LIN {X 0,Y 587.697,Z 859.31,A -85,B 0,C 180,E1 8837.447,E2 8837.447} C_VEL
LIN {X 0,Y 587.589,Z 859.31,A -85,B 0,C 180,E1 8842.753,E2 8842.753} C_VEL
LIN {X 0,Y 587.459,Z 859.31,A -85,B 0,C 180,E1 8847.659,E2 8847.659} C_VEL
LIN {X 0,Y 587.346,Z 859.31,A -85,B 0,C 180,E1 8852.797,E2 8852.797} C_VEL
LIN {X 0,Y 587.19,Z 859.31,A -85,B 0,C 180,E1 8858.258,E2 8858.258} C_VEL
LIN {X 0,Y 587.185,Z 859.31,A -85,B 0,C 180,E1 8864.156,E2 8864.156} C_VEL
LIN {X 0,Y 587.224,Z 859.31,A -85,B 0,C 180,E1 8869.826,E2 8869.826} C_VEL
LIN {X 0,Y 587.363,Z 859.919,A -85,B 0,C 180,E1 8871.339,E2 8871.339} C_VEL
LIN {X 0,Y 612.284,Z 916.303,A -85,B 0,C 180,E1 8873.785,E2 8873.785} C_VEL
LIN {X 0,Y 612.06,Z 926.776,A -85,B 0,C 180,E1 8873.959,E2 8873.959} C_VEL
LIN {X 0,Y 608.088,Z 943.76,A -85,B 0,C 180,E1 8874.115,E2 8874.115} C_VEL
LIN {X 0,Y 603.502,Z 960.575,A -85,B 0,C 180,E1 8874.323,E2 8874.323} C_VEL
LIN {X 0,Y 600.339,Z 1006.753,A -85,B 0,C 180,E1 8875.92,E2 8875.92} C_VEL
LIN {X 0,Y 596.482,Z 1051.642,A -85,B 0,C 180,E1 8878.158,E2 8878.158} C_VEL
LIN {X 0,Y 592.489,Z 1093.023,A -85,B 0,C 180,E1 8880.927,E2 8880.927} C_VEL
LIN {X 0,Y 588.871,Z 1128.661,A -85,B 0,C 180,E1 8884.059,E2 8884.059} C_VEL
LIN {X 0,Y 585.696,Z 1159.357,A -85,B 0,C 180,E1 8887.567,E2 8887.567} C_VEL
LIN {X 0,Y 583.284,Z 1184.333,A -85,B 0,C 180,E1 8891.257,E2 8891.257} C_VEL
LIN {X 0,Y 581.725,Z 1204.991,A -85,B 0,C 180,E1 8895.287,E2 8895.287} C_VEL
LIN {X 0,Y 580.827,Z 1221.162,A -85,B 0,C 180,E1 8899.857,E2 8899.857} C_VEL
LIN {X 0,Y 580.497,Z 1230.457,A -85,B 0,C 180,E1 8904.006,E2 8904.006} C_VEL
LIN {X 0,Y 580.504,Z 1235.164,A -85,B 0,C 180,E1 8908.504,E2 8908.504} C_VEL
LIN {X 0,Y 580.466,Z 1234.213,A -85,B 0,C 180,E1 8912.993,E2 8912.993} C_VEL
LIN {X 0,Y 580.544,Z 1229.327,A -85,B 0,C 180,E1 8916.683,E2 8916.683} C_VEL
LIN {X 0,Y 580.955,Z 1217.72,A -85,B 0,C 180,E1 8921.281,E2 8921.281} C_VEL
LIN {X 0,Y 582.016,Z 1201.38,A -85,B 0,C 180,E1 8925.504,E2 8925.504} C_VEL
LIN {X 0,Y 583.753,Z 1179.913,A -85,B 0,C 180,E1 8929.471,E2 8929.471} C_VEL
LIN {X 0,Y 586.43,Z 1151.644,A -85,B 0,C 180,E1 8933.414,E2 8933.414} C_VEL
LIN {X 0,Y 590.023,Z 1117.476,A -85,B 0,C 180,E1 8937.016,E2 8937.016} C_VEL
LIN {X 0,Y 594.013,Z 1078.354,A -85,B 0,C 180,E1 8940.148,E2 8940.148} C_VEL
LIN {X 0,Y 598.073,Z 1034.825,A -85,B 0,C 180,E1 8942.765,E2 8942.765} C_VEL
LIN {X 0,Y 601.694,Z 989.173,A -85,B 0,C 180,E1 8944.77,E2 8944.77} C_VEL
LIN {X 0,Y 604.598,Z 941.328,A -85,B 0,C 180,E1 8946.155,E2 8946.155} C_VEL
LIN {X 0,Y 605.195,Z 918.263,A -85,B 0,C 180,E1 8946.6,E2 8946.6} C_VEL
LIN {X 0,Y 583.541,Z 869.006,A -85,B 0,C 180,E1 8948.782,E2 8948.782} C_VEL
LIN {X 0,Y 579.403,Z 859.31,A -85,B 0,C 180,E1 8949.238,E2 8949.238} C_VEL
LIN {X 0,Y 579.376,Z 859.31,A -85,B 0,C 180,E1 8955.089,E2 8955.089} C_VEL
LIN {X 0,Y 579.271,Z 859.31,A -85,B 0,C 180,E1 8961.121,E2 8961.121} C_VEL
LIN {X 0,Y 579.379,Z 859.31,A -85,B 0,C 180,E1 8966.816,E2 8966.816} C_VEL
LIN {X 0,Y 579.578,Z 859.31,A -85,B 0,C 180,E1 8972.738,E2 8972.738} C_VEL
LIN {X 0,Y 579.689,Z 859.31,A -85,B 0,C 180,E1 8978.537,E2 8978.537} C_VEL
LIN {X 0,Y 579.76,Z 859.31,A -85,B 0,C 180,E1 8983.294,E2 8983.294} C_VEL
LIN {X 0,Y 579.901,Z 859.31,A -85,B 0,C 180,E1 8989.461,E2 8989.461} C_VEL
LIN {X 0,Y 580.104,Z 859.31,A -85,B 0,C 180,E1 8994.002,E2 8994.002} C_VEL
LIN {X 0,Y 580.244,Z 859.31,A -85,B 0,C 180,E1 8998.502,E2 8998.502} C_VEL
LIN {X 0,Y 580.215,Z 859.31,A -85,B 0,C 180,E1 9002.991,E2 9002.991} C_VEL
LIN {X 0,Y 580.045,Z 859.31,A -85,B 0,C 180,E1 9007.501,E2 9007.501} C_VEL
LIN {X 0,Y 579.905,Z 859.31,A -85,B 0,C 180,E1 9012.061,E2 9012.061} C_VEL
LIN {X 0,Y 579.803,Z 859.31,A -85,B 0,C 180,E1 9016.7,E2 9016.7} C_VEL
LIN {X 0,Y 579.663,Z 859.31,A -85,B 0,C 180,E1 9021.459,E2 9021.459} C_VEL
LIN {X 0,Y 579.514,Z 859.31,A -85,B 0,C 180,E1 9027.25,E2 9027.25} C_VEL
LIN {X 0,Y 579.386,Z 859.31,A -85,B 0,C 180,E1 9033.301,E2 9033.301} C_VEL
LIN {X 0,Y 579.282,Z 859.31,A -85,B 0,C 180,E1 9038.873,E2 9038.873} C_VEL
LIN {X 0,Y 579.235,Z 859.31,A -85,B 0,C 180,E1 9045.063,E2 9045.063} C_VEL
LIN {X 0,Y 579.333,Z 859.31,A -85,B 0,C 180,E1 9051.117,E2 9051.117} C_VEL
LIN {X 0,Y 579.475,Z 859.947,A -85,B 0,C 180,E1 9057.039,E2 9057.039} C_VEL
LIN {X 0,Y 604.152,Z 909.899,A -85,B 0,C 180,E1 9059.386,E2 9059.386} C_VEL
LIN {X 0,Y 603.053,Z 971.893,A -85,B 0,C 180,E1 9060.257,E2 9060.257} C_VEL
LIN {X 0,Y 600.509,Z 1012.044,A -85,B 0,C 180,E1 9061.399,E2 9061.399} C_VEL
LIN {X 0,Y 596.94,Z 1050.359,A -85,B 0,C 180,E1 9063.118,E2 9063.118} C_VEL
LIN {X 0,Y 592.943,Z 1085.359,A -85,B 0,C 180,E1 9065.354,E2 9065.354} C_VEL
LIN {X 0,Y 588.966,Z 1116.703,A -85,B 0,C 180,E1 9068.072,E2 9068.072} C_VEL
LIN {X 0,Y 585.696,Z 1143.269,A -85,B 0,C 180,E1 9071.138,E2 9071.138} C_VEL
LIN {X 0,Y 583.07,Z 1166.127,A -85,B 0,C 180,E1 9074.658,E2 9074.658} C_VEL
LIN {X 0,Y 581.532,Z 1183.649,A -85,B 0,C 180,E1 9078.35,E2 9078.35} C_VEL
LIN {X 0,Y 580.757,Z 1196.752,A -85,B 0,C 180,E1 9082.386,E2 9082.386} C_VEL
LIN {X 0,Y 580.526,Z 1203,A -85,B 0,C 180,E1 9085.509,E2 9085.509} C_VEL
LIN {X 0,Y 580.388,Z 1205.958,A -85,B 0,C 180,E1 9088.504,E2 9088.504} C_VEL
LIN {X 0,Y 580.489,Z 1205.894,A -85,B 0,C 180,E1 9091.496,E2 9091.496} C_VEL
LIN {X 0,Y 580.614,Z 1201.69,A -85,B 0,C 180,E1 9095.241,E2 9095.241} C_VEL
LIN {X 0,Y 580.972,Z 1191.508,A -85,B 0,C 180,E1 9099.382,E2 9099.382} C_VEL
LIN {X 0,Y 582.164,Z 1175.966,A -85,B 0,C 180,E1 9103.334,E2 9103.334} C_VEL
LIN {X 0,Y 584.19,Z 1155.887,A -85,B 0,C 180,E1 9106.966,E2 9106.966} C_VEL
LIN {X 0,Y 587.292,Z 1130.212,A -85,B 0,C 180,E1 9110.385,E2 9110.385} C_VEL
LIN {X 0,Y 591.008,Z 1100.781,A -85,B 0,C 180,E1 9113.316,E2 9113.316} C_VEL
LIN {X 0,Y 595.002,Z 1067.95,A -85,B 0,C 180,E1 9115.756,E2 9115.756} C_VEL
LIN {X 0,Y 598.679,Z 1033,A -85,B 0,C 180,E1 9117.652,E2 9117.652} C_VEL
LIN {X 0,Y 601.636,Z 995.563,A -85,B 0,C 180,E1 9119.055,E2 9119.055} C_VEL
LIN {X 0,Y 603.581,Z 956.066,A -85,B 0,C 180,E1 9119.942,E2 9119.942} C_VEL
LIN {X 0,Y 603.684,Z 908.974,A -85,B 0,C 180,E1 9120.562,E2 9120.562} C_VEL
LIN {X 0,Y 579.497,Z 860.059,A -85,B 0,C 180,E1 9122.861,E2 9122.861} C_VEL
LIN {X 0,Y 579.373,Z 859.31,A -85,B 0,C 180,E1 9128.337,E2 9128.337} C_VEL
LIN {X 0,Y 579.233,Z 859.31,A -85,B 0,C 180,E1 9132.924,E2 9132.924} C_VEL
LIN {X 0,Y 579.287,Z 859.31,A -85,B 0,C 180,E1 9139.176,E2 9139.176} C_VEL
LIN {X 0,Y 579.351,Z 859.31,A -85,B 0,C 180,E1 9144.885,E2 9144.885} C_VEL
LIN {X 0,Y 579.416,Z 859.31,A -85,B 0,C 180,E1 9150.217,E2 9150.217} C_VEL
LIN {X 0,Y 579.59,Z 859.31,A -85,B 0,C 180,E1 9155.282,E2 9155.282} C_VEL
LIN {X 0,Y 579.568,Z 859.31,A -85,B 0,C 180,E1 9160.259,E2 9160.259} C_VEL
LIN {X 0,Y 579.713,Z 859.31,A -85,B 0,C 180,E1 9166.4,E2 9166.4} C_VEL
LIN {X 0,Y 580.093,Z 859.31,A -85,B 0,C 180,E1 9172.169,E2 9172.169} C_VEL
LIN {X 0,Y 580.271,Z 859.31,A -85,B 0,C 180,E1 9177.009,E2 9177.009} C_VEL
LIN {X 0,Y 580.392,Z 859.31,A -85,B 0,C 180,E1 9181.498,E2 9181.498} C_VEL
LIN {X 0,Y 580.005,Z 859.31,A -85,B 0,C 180,E1 9186.893,E2 9186.893} C_VEL
LIN {X 0,Y 579.884,Z 859.31,A -85,B 0,C 180,E1 9192.065,E2 9192.065} C_VEL
LIN {X 0,Y 579.807,Z 859.31,A -85,B 0,C 180,E1 9196.705,E2 9196.705} C_VEL
LIN {X 0,Y 579.692,Z 859.31,A -85,B 0,C 180,E1 9201.463,E2 9201.463} C_VEL
LIN {X 0,Y 579.545,Z 859.31,A -85,B 0,C 180,E1 9207.255,E2 9207.255} C_VEL
LIN {X 0,Y 579.385,Z 859.31,A -85,B 0,C 180,E1 9213.306,E2 9213.306} C_VEL
LIN {X 0,Y 579.262,Z 859.31,A -85,B 0,C 180,E1 9218.88,E2 9218.88} C_VEL
LIN {X 0,Y 579.222,Z 859.31,A -85,B 0,C 180,E1 9225.062,E2 9225.062} C_VEL
LIN {X 0,Y 579.378,Z 859.31,A -85,B 0,C 180,E1 9230.754,E2 9230.754} C_VEL
LIN {X 0,Y 599.876,Z 906.09,A -85,B 0,C 180,E1 9232.87,E2 9232.87} C_VEL
LIN {X 0,Y 605.474,Z 920.812,A -85,B 0,C 180,E1 9233.461,E2 9233.461} C_VEL
LIN {X 0,Y 603.502,Z 960.575,A -85,B 0,C 180,E1 9234.323,E2 9234.323} C_VEL
LIN {X 0,Y 594.723,Z 991.691,A -85,B 0,C 180,E1 9234.944,E2 9234.944} C_VEL
LIN {X 0,Y 594.491,Z 993.669,A -85,B 0,C 180,E1 9235.019,E2 9235.019} C_VEL
LIN {X 0,Y 590.821,Z 1037.331,A -85,B 0,C 180,E1 9237.016,E2 9237.016} C_VEL
LIN {X 0,Y 586.644,Z 1078.873,A -85,B 0,C 180,E1 9239.595,E2 9239.595} C_VEL
LIN {X 0,Y 582.519,Z 1117.313,A -85,B 0,C 180,E1 9242.711,E2 9242.711} C_VEL
LIN {X 0,Y 578.817,Z 1151.567,A -85,B 0,C 180,E1 9246.357,E2 9246.357} C_VEL
LIN {X 0,Y 576.12,Z 1178.982,A -85,B 0,C 180,E1 9250.202,E2 9250.202} C_VEL
LIN {X 0,Y 574.243,Z 1200.385,A -85,B 0,C 180,E1 9254.154,E2 9254.154} C_VEL
LIN {X 0,Y 573.197,Z 1216.803,A -85,B 0,C 180,E1 9258.266,E2 9258.266} C_VEL
LIN {X 0,Y 572.66,Z 1227.634,A -85,B 0,C 180,E1 9262.397,E2 9262.397} C_VEL
LIN {X 0,Y 572.539,Z 1232.645,A -85,B 0,C 180,E1 9265.446,E2 9265.446} C_VEL
LIN {X 0,Y 572.567,Z 1235.5,A -85,B 0,C 180,E1 9270,E2 9270} C_VEL
LIN {X 0,Y 572.544,Z 1232.646,A -85,B 0,C 180,E1 9274.554,E2 9274.554} C_VEL
LIN {X 0,Y 572.685,Z 1226.068,A -85,B 0,C 180,E1 9278.368,E2 9278.368} C_VEL
LIN {X 0,Y 573.34,Z 1213.755,A -85,B 0,C 180,E1 9282.594,E2 9282.594} C_VEL
LIN {X 0,Y 574.504,Z 1196.74,A -85,B 0,C 180,E1 9286.612,E2 9286.612} C_VEL
LIN {X 0,Y 576.593,Z 1172.554,A -85,B 0,C 180,E1 9290.809,E2 9290.809} C_VEL
LIN {X 0,Y 579.67,Z 1143.649,A -85,B 0,C 180,E1 9294.568,E2 9294.568} C_VEL
LIN {X 0,Y 583.082,Z 1111.739,A -85,B 0,C 180,E1 9297.785,E2 9297.785} C_VEL
LIN {X 0,Y 587.072,Z 1074.285,A -85,B 0,C 180,E1 9300.722,E2 9300.722} C_VEL
LIN {X 0,Y 591.139,Z 1033.204,A -85,B 0,C 180,E1 9303.206,E2 9303.206} C_VEL
LIN {X 0,Y 594.921,Z 988.204,A -85,B 0,C 180,E1 9305.191,E2 9305.191} C_VEL
LIN {X 0,Y 597.93,Z 940.993,A -85,B 0,C 180,E1 9306.564,E2 9306.564} C_VEL
LIN {X 0,Y 598.169,Z 920.224,A -85,B 0,C 180,E1 9306.997,E2 9306.997} C_VEL
LIN {X 0,Y 577.934,Z 873.583,A -85,B 0,C 180,E1 9309.102,E2 9309.102} C_VEL
LIN {X 0,Y 571.434,Z 859.31,A -85,B 0,C 180,E1 9309.855,E2 9309.855} C_VEL
LIN {X 0,Y 571.382,Z 859.31,A -85,B 0,C 180,E1 9315.728,E2 9315.728} C_VEL
LIN {X 0,Y 571.327,Z 859.31,A -85,B 0,C 180,E1 9320.476,E2 9320.476} C_VEL
LIN {X 0,Y 571.383,Z 859.31,A -85,B 0,C 180,E1 9326.165,E2 9326.165} C_VEL
LIN {X 0,Y 571.588,Z 859.31,A -85,B 0,C 180,E1 9331.504,E2 9331.504} C_VEL
LIN {X 0,Y 571.752,Z 859.31,A -85,B 0,C 180,E1 9336.58,E2 9336.58} C_VEL
LIN {X 0,Y 571.821,Z 859.31,A -85,B 0,C 180,E1 9342.549,E2 9342.549} C_VEL
LIN {X 0,Y 571.928,Z 859.31,A -85,B 0,C 180,E1 9348.606,E2 9348.606} C_VEL
LIN {X 0,Y 572.205,Z 859.31,A -85,B 0,C 180,E1 9353.919,E2 9353.919} C_VEL
LIN {X 0,Y 572.342,Z 859.31,A -85,B 0,C 180,E1 9358.481,E2 9358.481} C_VEL
LIN {X 0,Y 572.314,Z 859.31,A -85,B 0,C 180,E1 9363.033,E2 9363.033} C_VEL
LIN {X 0,Y 572.127,Z 859.31,A -85,B 0,C 180,E1 9367.606,E2 9367.606} C_VEL
LIN {X 0,Y 571.984,Z 859.31,A -85,B 0,C 180,E1 9372.23,E2 9372.23} C_VEL
LIN {X 0,Y 571.829,Z 859.31,A -85,B 0,C 180,E1 9377.453,E2 9377.453} C_VEL
LIN {X 0,Y 571.699,Z 859.31,A -85,B 0,C 180,E1 9383.418,E2 9383.418} C_VEL
LIN {X 0,Y 571.54,Z 859.31,A -85,B 0,C 180,E1 9388.966,E2 9388.966} C_VEL
LIN {X 0,Y 571.392,Z 859.31,A -85,B 0,C 180,E1 9394.705,E2 9394.705} C_VEL
LIN {X 0,Y 571.309,Z 859.31,A -85,B 0,C 180,E1 9399.721,E2 9399.721} C_VEL
LIN {X 0,Y 571.258,Z 859.31,A -85,B 0,C 180,E1 9405.722,E2 9405.722} C_VEL
LIN {X 0,Y 571.349,Z 859.31,A -85,B 0,C 180,E1 9410.468,E2 9410.468} C_VEL
LIN {X 0,Y 571.475,Z 859.31,A -85,B 0,C 180,E1 9416.435,E2 9416.435} C_VEL
LIN {X 0,Y 578.232,Z 873.768,A -85,B 0,C 180,E1 9417.136,E2 9417.136} C_VEL
LIN {X 0,Y 597.673,Z 913.926,A -85,B 0,C 180,E1 9419.013,E2 9419.013} C_VEL
LIN {X 0,Y 596.487,Z 971.573,A -85,B 0,C 180,E1 9419.832,E2 9419.832} C_VEL
LIN {X 0,Y 593.767,Z 1012.202,A -85,B 0,C 180,E1 9420.996,E2 9420.996} C_VEL
LIN {X 0,Y 590.145,Z 1049.593,A -85,B 0,C 180,E1 9422.68,E2 9422.68} C_VEL
LIN {X 0,Y 585.912,Z 1084.949,A -85,B 0,C 180,E1 9424.945,E2 9424.945} C_VEL
LIN {X 0,Y 581.693,Z 1116.6,A -85,B 0,C 180,E1 9427.708,E2 9427.708} C_VEL
LIN {X 0,Y 578.142,Z 1143.832,A -85,B 0,C 180,E1 9430.887,E2 9430.887} C_VEL
LIN {X 0,Y 575.352,Z 1166.873,A -85,B 0,C 180,E1 9434.493,E2 9434.493} C_VEL
LIN {X 0,Y 573.743,Z 1184.091,A -85,B 0,C 180,E1 9438.189,E2 9438.189} C_VEL
LIN {X 0,Y 573.01,Z 1195.446,A -85,B 0,C 180,E1 9441.637,E2 9441.637} C_VEL
LIN {X 0,Y 572.663,Z 1203.237,A -85,B 0,C 180,E1 9445.447,E2 9445.447} C_VEL
LIN {X 0,Y 572.506,Z 1206.164,A -85,B 0,C 180,E1 9448.484,E2 9448.484} C_VEL
LIN {X 0,Y 572.62,Z 1206.103,A -85,B 0,C 180,E1 9451.517,E2 9451.517} C_VEL
LIN {X 0,Y 572.731,Z 1201.943,A -85,B 0,C 180,E1 9455.313,E2 9455.313} C_VEL
LIN {X 0,Y 573.136,Z 1191.887,A -85,B 0,C 180,E1 9459.511,E2 9459.511} C_VEL
LIN {X 0,Y 574.369,Z 1177.169,A -85,B 0,C 180,E1 9463.371,E2 9463.371} C_VEL
LIN {X 0,Y 576.586,Z 1156.417,A -85,B 0,C 180,E1 9467.197,E2 9467.197} C_VEL
LIN {X 0,Y 579.852,Z 1130.793,A -85,B 0,C 180,E1 9470.658,E2 9470.658} C_VEL
LIN {X 0,Y 583.768,Z 1101.465,A -85,B 0,C 180,E1 9473.623,E2 9473.623} C_VEL
LIN {X 0,Y 587.928,Z 1068.798,A -85,B 0,C 180,E1 9476.089,E2 9476.089} C_VEL
LIN {X 0,Y 591.882,Z 1033.144,A -85,B 0,C 180,E1 9478.046,E2 9478.046} C_VEL
LIN {X 0,Y 594.997,Z 995.399,A -85,B 0,C 180,E1 9479.473,E2 9479.473} C_VEL
LIN {X 0,Y 597.042,Z 954.642,A -85,B 0,C 180,E1 9480.384,E2 9480.384} C_VEL
LIN {X 0,Y 597.195,Z 911.71,A -85,B 0,C 180,E1 9480.953,E2 9480.953} C_VEL
LIN {X 0,Y 571.691,Z 860.878,A -85,B 0,C 180,E1 9483.428,E2 9483.428} C_VEL
LIN {X 0,Y 571.494,Z 859.31,A -85,B 0,C 180,E1 9483.51,E2 9483.51} C_VEL
LIN {X 0,Y 571.468,Z 859.31,A -85,B 0,C 180,E1 9487.58,E2 9487.58} C_VEL
LIN {X 0,Y 571.272,Z 859.31,A -85,B 0,C 180,E1 9493.602,E2 9493.602} C_VEL
LIN {X 0,Y 571.286,Z 859.31,A -85,B 0,C 180,E1 9498.479,E2 9498.479} C_VEL
LIN {X 0,Y 571.455,Z 859.31,A -85,B 0,C 180,E1 9504.326,E2 9504.326} C_VEL
LIN {X 0,Y 571.52,Z 859.31,A -85,B 0,C 180,E1 9509.763,E2 9509.763} C_VEL
LIN {X 0,Y 571.638,Z 859.31,A -85,B 0,C 180,E1 9514.914,E2 9514.914} C_VEL
LIN {X 0,Y 571.662,Z 859.31,A -85,B 0,C 180,E1 9519.851,E2 9519.851} C_VEL
LIN {X 0,Y 571.812,Z 859.31,A -85,B 0,C 180,E1 9526.208,E2 9526.208} C_VEL
LIN {X 0,Y 572.191,Z 859.31,A -85,B 0,C 180,E1 9532.184,E2 9532.184} C_VEL
LIN {X 0,Y 572.364,Z 859.31,A -85,B 0,C 180,E1 9536.968,E2 9536.968} C_VEL
LIN {X 0,Y 572.486,Z 859.31,A -85,B 0,C 180,E1 9541.518,E2 9541.518} C_VEL
LIN {X 0,Y 572.229,Z 859.31,A -85,B 0,C 180,E1 9546.081,E2 9546.081} C_VEL
LIN {X 0,Y 571.968,Z 859.31,A -85,B 0,C 180,E1 9552.235,E2 9552.235} C_VEL
LIN {X 0,Y 571.863,Z 859.31,A -85,B 0,C 180,E1 9557.463,E2 9557.463} C_VEL
LIN {X 0,Y 571.725,Z 859.31,A -85,B 0,C 180,E1 9563.421,E2 9563.421} C_VEL
LIN {X 0,Y 571.568,Z 859.31,A -85,B 0,C 180,E1 9568.97,E2 9568.97} C_VEL
LIN {X 0,Y 571.396,Z 859.31,A -85,B 0,C 180,E1 9574.705,E2 9574.705} C_VEL
LIN {X 0,Y 571.306,Z 859.31,A -85,B 0,C 180,E1 9579.72,E2 9579.72} C_VEL
LIN {X 0,Y 571.249,Z 859.31,A -85,B 0,C 180,E1 9585.729,E2 9585.729} C_VEL
LIN {X 0,Y 571.412,Z 859.519,A -85,B 0,C 180,E1 9590.2,E2 9590.2} C_VEL
LIN {X 0,Y 591.691,Z 904.574,A -85,B 0,C 180,E1 9592.325,E2 9592.325} C_VEL
LIN {X 0,Y 598.794,Z 921.954,A -85,B 0,C 180,E1 9593.074,E2 9593.074} C_VEL
LIN {X 0,Y 596.308,Z 967.89,A -85,B 0,C 180,E1 9594.141,E2 9594.141} C_VEL
LIN {X 0,Y 594.491,Z 993.669,A -85,B 0,C 180,E1 9595.019,E2 9595.019} C_VEL
LIN {X 0,Y 589.837,Z 1009.893,A -85,B 0,C 180,E1 9595.494,E2 9595.494} C_VEL
LIN {X 0,Y 584.927,Z 1025.72,A -85,B 0,C 180,E1 9596.04,E2 9596.04} C_VEL
LIN {X 0,Y 580.78,Z 1065.697,A -85,B 0,C 180,E1 9598.347,E2 9598.347} C_VEL
LIN {X 0,Y 576.433,Z 1104.91,A -85,B 0,C 180,E1 9601.331,E2 9601.331} C_VEL
LIN {X 0,Y 572.4,Z 1140.312,A -85,B 0,C 180,E1 9604.812,E2 9604.812} C_VEL
LIN {X 0,Y 569.079,Z 1170.554,A -85,B 0,C 180,E1 9608.707,E2 9608.707} C_VEL
LIN {X 0,Y 566.932,Z 1192.958,A -85,B 0,C 180,E1 9612.501,E2 9612.501} C_VEL
LIN {X 0,Y 565.581,Z 1210.591,A -85,B 0,C 180,E1 9616.442,E2 9616.442} C_VEL
LIN {X 0,Y 564.936,Z 1224.024,A -85,B 0,C 180,E1 9620.739,E2 9620.739} C_VEL
LIN {X 0,Y 564.773,Z 1231.666,A -85,B 0,C 180,E1 9624.611,E2 9624.611} C_VEL
LIN {X 0,Y 564.705,Z 1235.164,A -85,B 0,C 180,E1 9628.462,E2 9628.462} C_VEL
LIN {X 0,Y 564.655,Z 1234.212,A -85,B 0,C 180,E1 9633.076,E2 9633.076} C_VEL
LIN {X 0,Y 564.736,Z 1229.042,A -85,B 0,C 180,E1 9636.997,E2 9636.997} C_VEL
LIN {X 0,Y 565.244,Z 1217.812,A -85,B 0,C 180,E1 9641.466,E2 9641.466} C_VEL
LIN {X 0,Y 566.292,Z 1201.984,A -85,B 0,C 180,E1 9645.619,E2 9645.619} C_VEL
LIN {X 0,Y 568.129,Z 1180.903,A -85,B 0,C 180,E1 9649.678,E2 9649.678} C_VEL
LIN {X 0,Y 570.958,Z 1152.741,A -85,B 0,C 180,E1 9653.714,E2 9653.714} C_VEL
LIN {X 0,Y 574.663,Z 1120.216,A -85,B 0,C 180,E1 9657.268,E2 9657.268} C_VEL
LIN {X 0,Y 578.825,Z 1083.042,A -85,B 0,C 180,E1 9660.424,E2 9660.424} C_VEL
LIN {X 0,Y 583.013,Z 1044.183,A -85,B 0,C 180,E1 9662.977,E2 9662.977} C_VEL
LIN {X 0,Y 586.998,Z 1002.566,A -85,B 0,C 180,E1 9665.025,E2 9665.025} C_VEL
LIN {X 0,Y 590.465,Z 957.258,A -85,B 0,C 180,E1 9666.57,E2 9666.57} C_VEL
LIN {X 0,Y 591.537,Z 922.812,A -85,B 0,C 180,E1 9667.371,E2 9667.371} C_VEL
LIN {X 0,Y 572.442,Z 878.305,A -85,B 0,C 180,E1 9669.419,E2 9669.419} C_VEL
LIN {X 0,Y 563.55,Z 859.31,A -85,B 0,C 180,E1 9670.446,E2 9670.446} C_VEL
LIN {X 0,Y 563.468,Z 859.31,A -85,B 0,C 180,E1 9676.559,E2 9676.559} C_VEL
LIN {X 0,Y 563.371,Z 859.31,A -85,B 0,C 180,E1 9681.793,E2 9681.793} C_VEL
LIN {X 0,Y 563.512,Z 859.31,A -85,B 0,C 180,E1 9687.473,E2 9687.473} C_VEL
LIN {X 0,Y 563.718,Z 859.31,A -85,B 0,C 180,E1 9692.814,E2 9692.814} C_VEL
LIN {X 0,Y 563.845,Z 859.31,A -85,B 0,C 180,E1 9697.903,E2 9697.903} C_VEL
LIN {X 0,Y 563.943,Z 859.31,A -85,B 0,C 180,E1 9702.811,E2 9702.811} C_VEL
LIN {X 0,Y 564.086,Z 859.31,A -85,B 0,C 180,E1 9709.162,E2 9709.162} C_VEL
LIN {X 0,Y 564.292,Z 859.31,A -85,B 0,C 180,E1 9713.833,E2 9713.833} C_VEL
LIN {X 0,Y 564.44,Z 859.31,A -85,B 0,C 180,E1 9718.46,E2 9718.46} C_VEL
LIN {X 0,Y 564.41,Z 859.31,A -85,B 0,C 180,E1 9723.075,E2 9723.075} C_VEL
LIN {X 0,Y 564.231,Z 859.31,A -85,B 0,C 180,E1 9727.713,E2 9727.713} C_VEL
LIN {X 0,Y 564.059,Z 859.31,A -85,B 0,C 180,E1 9732.405,E2 9732.405} C_VEL
LIN {X 0,Y 563.965,Z 859.31,A -85,B 0,C 180,E1 9737.184,E2 9737.184} C_VEL
LIN {X 0,Y 563.811,Z 859.31,A -85,B 0,C 180,E1 9742.094,E2 9742.094} C_VEL
LIN {X 0,Y 563.625,Z 859.31,A -85,B 0,C 180,E1 9747.477,E2 9747.477} C_VEL
LIN {X 0,Y 563.512,Z 859.31,A -85,B 0,C 180,E1 9752.522,E2 9752.522} C_VEL
LIN {X 0,Y 563.394,Z 859.31,A -85,B 0,C 180,E1 9758.199,E2 9758.199} C_VEL
LIN {X 0,Y 563.37,Z 859.31,A -85,B 0,C 180,E1 9763.43,E2 9763.43} C_VEL
LIN {X 0,Y 563.374,Z 859.31,A -85,B 0,C 180,E1 9768.84,E2 9768.84} C_VEL
LIN {X 0,Y 563.512,Z 859.31,A -85,B 0,C 180,E1 9773.751,E2 9773.751} C_VEL
LIN {X 0,Y 563.549,Z 859.31,A -85,B 0,C 180,E1 9775.812,E2 9775.812} C_VEL
LIN {X 0,Y 568.333,Z 869.711,A -85,B 0,C 180,E1 9776.343,E2 9776.343} C_VEL
LIN {X 0,Y 591.167,Z 915.978,A -85,B 0,C 180,E1 9778.604,E2 9778.604} C_VEL
LIN {X 0,Y 589.9,Z 972.039,A -85,B 0,C 180,E1 9779.417,E2 9779.417} C_VEL
LIN {X 0,Y 587.114,Z 1011.651,A -85,B 0,C 180,E1 9780.557,E2 9780.557} C_VEL
LIN {X 0,Y 583.2,Z 1050.448,A -85,B 0,C 180,E1 9782.327,E2 9782.327} C_VEL
LIN {X 0,Y 578.771,Z 1085.611,A -85,B 0,C 180,E1 9784.614,E2 9784.614} C_VEL
LIN {X 0,Y 574.425,Z 1116.758,A -85,B 0,C 180,E1 9787.368,E2 9787.368} C_VEL
LIN {X 0,Y 570.565,Z 1144.617,A -85,B 0,C 180,E1 9790.669,E2 9790.669} C_VEL
LIN {X 0,Y 567.653,Z 1167.512,A -85,B 0,C 180,E1 9794.322,E2 9794.322} C_VEL
LIN {X 0,Y 565.946,Z 1184.458,A -85,B 0,C 180,E1 9798.024,E2 9798.024} C_VEL
LIN {X 0,Y 565.137,Z 1195.773,A -85,B 0,C 180,E1 9801.52,E2 9801.52} C_VEL
LIN {X 0,Y 564.772,Z 1203.482,A -85,B 0,C 180,E1 9805.383,E2 9805.383} C_VEL
LIN {X 0,Y 564.608,Z 1206.371,A -85,B 0,C 180,E1 9808.462,E2 9808.462} C_VEL
LIN {X 0,Y 564.72,Z 1206.31,A -85,B 0,C 180,E1 9811.538,E2 9811.538} C_VEL
LIN {X 0,Y 564.852,Z 1202.194,A -85,B 0,C 180,E1 9815.388,E2 9815.388} C_VEL
LIN {X 0,Y 565.324,Z 1192.233,A -85,B 0,C 180,E1 9819.644,E2 9819.644} C_VEL
LIN {X 0,Y 566.591,Z 1177.66,A -85,B 0,C 180,E1 9823.534,E2 9823.534} C_VEL
LIN {X 0,Y 568.964,Z 1156.872,A -85,B 0,C 180,E1 9827.435,E2 9827.435} C_VEL
LIN {X 0,Y 572.42,Z 1131.322,A -85,B 0,C 180,E1 9830.939,E2 9830.939} C_VEL
LIN {X 0,Y 576.676,Z 1100.976,A -85,B 0,C 180,E1 9834.034,E2 9834.034} C_VEL
LIN {X 0,Y 581.073,Z 1068.091,A -85,B 0,C 180,E1 9836.525,E2 9836.525} C_VEL
LIN {X 0,Y 585.049,Z 1033.737,A -85,B 0,C 180,E1 9838.428,E2 9838.428} C_VEL
LIN {X 0,Y 588.365,Z 995.375,A -85,B 0,C 180,E1 9839.894,E2 9839.894} C_VEL
LIN {X 0,Y 590.493,Z 955.748,A -85,B 0,C 180,E1 9840.797,E2 9840.797} C_VEL
LIN {X 0,Y 590.602,Z 914.164,A -85,B 0,C 180,E1 9841.363,E2 9841.363} C_VEL
LIN {X 0,Y 563.561,Z 859.31,A -85,B 0,C 180,E1 9844.108,E2 9844.108} C_VEL
LIN {X 0,Y 563.394,Z 859.31,A -85,B 0,C 180,E1 9850.203,E2 9850.203} C_VEL
LIN {X 0,Y 563.363,Z 859.31,A -85,B 0,C 180,E1 9855.645,E2 9855.645} C_VEL
LIN {X 0,Y 563.414,Z 859.31,A -85,B 0,C 180,E1 9861.802,E2 9861.802} C_VEL
LIN {X 0,Y 563.524,Z 859.31,A -85,B 0,C 180,E1 9867.479,E2 9867.479} C_VEL
LIN {X 0,Y 563.655,Z 859.31,A -85,B 0,C 180,E1 9872.815,E2 9872.815} C_VEL
LIN {X 0,Y 563.795,Z 859.31,A -85,B 0,C 180,E1 9877.905,E2 9877.905} C_VEL
LIN {X 0,Y 563.738,Z 859.31,A -85,B 0,C 180,E1 9882.809,E2 9882.809} C_VEL
LIN {X 0,Y 564.011,Z 859.31,A -85,B 0,C 180,E1 9887.594,E2 9887.594} C_VEL
LIN {X 0,Y 564.312,Z 859.31,A -85,B 0,C 180,E1 9893.478,E2 9893.478} C_VEL
LIN {X 0,Y 564.443,Z 859.31,A -85,B 0,C 180,E1 9898.464,E2 9898.464} C_VEL
LIN {X 0,Y 564.411,Z 859.31,A -85,B 0,C 180,E1 9903.079,E2 9903.079} C_VEL
LIN {X 0,Y 564.193,Z 859.31,A -85,B 0,C 180,E1 9907.718,E2 9907.718} C_VEL
LIN {X 0,Y 564.044,Z 859.31,A -85,B 0,C 180,E1 9912.41,E2 9912.41} C_VEL
LIN {X 0,Y 563.985,Z 859.31,A -85,B 0,C 180,E1 9917.188,E2 9917.188} C_VEL
LIN {X 0,Y 563.84,Z 859.31,A -85,B 0,C 180,E1 9922.097,E2 9922.097} C_VEL
LIN {X 0,Y 563.656,Z 859.31,A -85,B 0,C 180,E1 9927.482,E2 9927.482} C_VEL
LIN {X 0,Y 563.523,Z 859.31,A -85,B 0,C 180,E1 9932.526,E2 9932.526} C_VEL
LIN {X 0,Y 563.372,Z 859.31,A -85,B 0,C 180,E1 9938.207,E2 9938.207} C_VEL
LIN {X 0,Y 563.363,Z 859.31,A -85,B 0,C 180,E1 9943.429,E2 9943.429} C_VEL
LIN {X 0,Y 563.493,Z 859.31,A -85,B 0,C 180,E1 9949.582,E2 9949.582} C_VEL
LIN {X 0,Y 574.222,Z 882.038,A -85,B 0,C 180,E1 9950.774,E2 9950.774} C_VEL
LIN {X 0,Y 592.066,Z 923.859,A -85,B 0,C 180,E1 9952.684,E2 9952.684} C_VEL
LIN {X 0,Y 589.333,Z 972.028,A -85,B 0,C 180,E1 9953.857,E2 9953.857} C_VEL
LIN {X 0,Y 585.743,Z 1017.336,A -85,B 0,C 180,E1 9955.633,E2 9955.633} C_VEL
LIN {X 0,Y 584.927,Z 1025.72,A -85,B 0,C 180,E1 9956.04,E2 9956.04} C_VEL
LIN {X 0,Y 579.669,Z 1041.333,A -85,B 0,C 180,E1 9956.663,E2 9956.663} C_VEL
LIN {X 0,Y 574.926,Z 1054.585,A -85,B 0,C 180,E1 9957.265,E2 9957.265} C_VEL
LIN {X 0,Y 574.692,Z 1056.395,A -85,B 0,C 180,E1 9957.379,E2 9957.379} C_VEL
LIN {X 0,Y 570.243,Z 1094.326,A -85,B 0,C 180,E1 9960.116,E2 9960.116} C_VEL
LIN {X 0,Y 566.016,Z 1130.101,A -85,B 0,C 180,E1 9963.456,E2 9963.456} C_VEL
LIN {X 0,Y 562.429,Z 1161.484,A -85,B 0,C 180,E1 9967.214,E2 9967.214} C_VEL
LIN {X 0,Y 559.63,Z 1187.68,A -85,B 0,C 180,E1 9971.346,E2 9971.346} C_VEL
LIN {X 0,Y 557.998,Z 1207.077,A -85,B 0,C 180,E1 9975.459,E2 9975.459} C_VEL
LIN {X 0,Y 557.157,Z 1221.761,A -85,B 0,C 180,E1 9979.818,E2 9979.818} C_VEL
LIN {X 0,Y 556.873,Z 1231.455,A -85,B 0,C 180,E1 9984.535,E2 9984.535} C_VEL
LIN {X 0,Y 556.8,Z 1235.035,A -85,B 0,C 180,E1 9988.44,E2 9988.44} C_VEL
LIN {X 0,Y 556.77,Z 1234.061,A -85,B 0,C 180,E1 9993.12,E2 9993.12} C_VEL
LIN {X 0,Y 556.828,Z 1228.788,A -85,B 0,C 180,E1 9997.097,E2 9997.097} C_VEL
LIN {X 0,Y 557.357,Z 1217.988,A -85,B 0,C 180,E1 10001.463,E2 10001.463} C_VEL
LIN {X 0,Y 558.457,Z 1202.005,A -85,B 0,C 180,E1 10005.744,E2 10005.744} C_VEL
LIN {X 0,Y 560.466,Z 1180.213,A -85,B 0,C 180,E1 10009.958,E2 10009.958} C_VEL
LIN {X 0,Y 563.543,Z 1151.237,A -85,B 0,C 180,E1 10014.128,E2 10014.128} C_VEL
LIN {X 0,Y 567.588,Z 1116.917,A -85,B 0,C 180,E1 10017.878,E2 10017.878} C_VEL
LIN {X 0,Y 572.307,Z 1077.495,A -85,B 0,C 180,E1 10021.195,E2 10021.195} C_VEL
LIN {X 0,Y 576.942,Z 1036.005,A -85,B 0,C 180,E1 10023.828,E2 10023.828} C_VEL
LIN {X 0,Y 581.229,Z 990.397,A -85,B 0,C 180,E1 10025.924,E2 10025.924} C_VEL
LIN {X 0,Y 584.658,Z 941.744,A -85,B 0,C 180,E1 10027.387,E2 10027.387} C_VEL
LIN {X 0,Y 585.031,Z 925.7,A -85,B 0,C 180,E1 10027.742,E2 10027.742} C_VEL
LIN {X 0,Y 567.748,Z 884.732,A -85,B 0,C 180,E1 10029.657,E2 10029.657} C_VEL
LIN {X 0,Y 555.601,Z 859.31,A -85,B 0,C 180,E1 10031.037,E2 10031.037} C_VEL
LIN {X 0,Y 555.564,Z 859.31,A -85,B 0,C 180,E1 10037.021,E2 10037.021} C_VEL
LIN {X 0,Y 555.439,Z 859.31,A -85,B 0,C 180,E1 10043.126,E2 10043.126} C_VEL
LIN {X 0,Y 555.632,Z 859.31,A -85,B 0,C 180,E1 10048.798,E2 10048.798} C_VEL
LIN {X 0,Y 555.819,Z 859.31,A -85,B 0,C 180,E1 10054.143,E2 10054.143} C_VEL
LIN {X 0,Y 555.935,Z 859.31,A -85,B 0,C 180,E1 10059.251,E2 10059.251} C_VEL
LIN {X 0,Y 556.026,Z 859.31,A -85,B 0,C 180,E1 10064.188,E2 10064.188} C_VEL
LIN {X 0,Y 556.159,Z 859.31,A -85,B 0,C 180,E1 10069.006,E2 10069.006} C_VEL
LIN {X 0,Y 556.406,Z 859.31,A -85,B 0,C 180,E1 10073.746,E2 10073.746} C_VEL
LIN {X 0,Y 556.544,Z 859.31,A -85,B 0,C 180,E1 10078.438,E2 10078.438} C_VEL
LIN {X 0,Y 556.514,Z 859.31,A -85,B 0,C 180,E1 10083.119,E2 10083.119} C_VEL
LIN {X 0,Y 556.31,Z 859.31,A -85,B 0,C 180,E1 10087.823,E2 10087.823} C_VEL
LIN {X 0,Y 556.163,Z 859.31,A -85,B 0,C 180,E1 10092.584,E2 10092.584} C_VEL
LIN {X 0,Y 556.022,Z 859.31,A -85,B 0,C 180,E1 10097.479,E2 10097.479} C_VEL
LIN {X 0,Y 555.883,Z 859.31,A -85,B 0,C 180,E1 10102.426,E2 10102.426} C_VEL
LIN {X 0,Y 555.72,Z 859.31,A -85,B 0,C 180,E1 10107.606,E2 10107.606} C_VEL
LIN {X 0,Y 555.595,Z 859.31,A -85,B 0,C 180,E1 10113.044,E2 10113.044} C_VEL
LIN {X 0,Y 555.492,Z 859.31,A -85,B 0,C 180,E1 10118.844,E2 10118.844} C_VEL
LIN {X 0,Y 555.442,Z 859.31,A -85,B 0,C 180,E1 10124.822,E2 10124.822} C_VEL
LIN {X 0,Y 555.535,Z 859.31,A -85,B 0,C 180,E1 10131.145,E2 10131.145} C_VEL
LIN {X 0,Y 555.566,Z 859.31,A -85,B 0,C 180,E1 10135.167,E2 10135.167} C_VEL
LIN {X 0,Y 562.808,Z 874.26,A -85,B 0,C 180,E1 10135.982,E2 10135.982} C_VEL
LIN {X 0,Y 584.688,Z 918.038,A -85,B 0,C 180,E1 10138.187,E2 10138.187} C_VEL
LIN {X 0,Y 583.36,Z 972.174,A -85,B 0,C 180,E1 10138.987,E2 10138.987} C_VEL
LIN {X 0,Y 580.448,Z 1011.501,A -85,B 0,C 180,E1 10140.126,E2 10140.126} C_VEL
LIN {X 0,Y 576.469,Z 1049.594,A -85,B 0,C 180,E1 10141.868,E2 10141.868} C_VEL
LIN {X 0,Y 571.91,Z 1084.427,A -85,B 0,C 180,E1 10144.133,E2 10144.133} C_VEL
LIN {X 0,Y 567.298,Z 1116.19,A -85,B 0,C 180,E1 10146.947,E2 10146.947} C_VEL
LIN {X 0,Y 563.289,Z 1143.365,A -85,B 0,C 180,E1 10150.164,E2 10150.164} C_VEL
LIN {X 0,Y 560.133,Z 1166.851,A -85,B 0,C 180,E1 10153.907,E2 10153.907} C_VEL
LIN {X 0,Y 558.166,Z 1184.727,A -85,B 0,C 180,E1 10157.842,E2 10157.842} C_VEL
LIN {X 0,Y 557.267,Z 1196.054,A -85,B 0,C 180,E1 10161.399,E2 10161.399} C_VEL
LIN {X 0,Y 556.908,Z 1203.713,A -85,B 0,C 180,E1 10165.318,E2 10165.318} C_VEL
LIN {X 0,Y 556.711,Z 1206.577,A -85,B 0,C 180,E1 10168.44,E2 10168.44} C_VEL
LIN {X 0,Y 556.82,Z 1206.517,A -85,B 0,C 180,E1 10171.56,E2 10171.56} C_VEL
LIN {X 0,Y 556.958,Z 1202.432,A -85,B 0,C 180,E1 10175.464,E2 10175.464} C_VEL
LIN {X 0,Y 557.48,Z 1192.525,A -85,B 0,C 180,E1 10179.781,E2 10179.781} C_VEL
LIN {X 0,Y 558.839,Z 1177.996,A -85,B 0,C 180,E1 10183.725,E2 10183.725} C_VEL
LIN {X 0,Y 561.359,Z 1157.287,A -85,B 0,C 180,E1 10187.679,E2 10187.679} C_VEL
LIN {X 0,Y 564.992,Z 1131.808,A -85,B 0,C 180,E1 10191.227,E2 10191.227} C_VEL
LIN {X 0,Y 569.457,Z 1101.569,A -85,B 0,C 180,E1 10194.359,E2 10194.359} C_VEL
LIN {X 0,Y 574.047,Z 1068.849,A -85,B 0,C 180,E1 10196.875,E2 10196.875} C_VEL
LIN {X 0,Y 578.372,Z 1032.867,A -85,B 0,C 180,E1 10198.884,E2 10198.884} C_VEL
LIN {X 0,Y 581.732,Z 995.606,A -85,B 0,C 180,E1 10200.318,E2 10200.318} C_VEL
LIN {X 0,Y 583.983,Z 956.673,A -85,B 0,C 180,E1 10201.22,E2 10201.22} C_VEL
LIN {X 0,Y 584.004,Z 916.605,A -85,B 0,C 180,E1 10201.785,E2 10201.785} C_VEL
LIN {X 0,Y 556.8,Z 863.468,A -85,B 0,C 180,E1 10204.549,E2 10204.549} C_VEL
LIN {X 0,Y 555.584,Z 859.31,A -85,B 0,C 180,E1 10204.802,E2 10204.802} C_VEL
LIN {X 0,Y 555.481,Z 859.31,A -85,B 0,C 180,E1 10210.897,E2 10210.897} C_VEL
LIN {X 0,Y 555.446,Z 859.31,A -85,B 0,C 180,E1 10217.016,E2 10217.016} C_VEL
LIN {X 0,Y 555.506,Z 859.31,A -85,B 0,C 180,E1 10223.136,E2 10223.136} C_VEL
LIN {X 0,Y 555.62,Z 859.31,A -85,B 0,C 180,E1 10228.802,E2 10228.802} C_VEL
LIN {X 0,Y 555.76,Z 859.31,A -85,B 0,C 180,E1 10234.145,E2 10234.145} C_VEL
LIN {X 0,Y 555.833,Z 859.31,A -85,B 0,C 180,E1 10239.251,E2 10239.251} C_VEL
LIN {X 0,Y 555.836,Z 859.31,A -85,B 0,C 180,E1 10244.187,E2 10244.187} C_VEL
LIN {X 0,Y 556.188,Z 859.31,A -85,B 0,C 180,E1 10249.011,E2 10249.011} C_VEL
LIN {X 0,Y 556.435,Z 859.31,A -85,B 0,C 180,E1 10253.75,E2 10253.75} C_VEL
LIN {X 0,Y 556.547,Z 859.31,A -85,B 0,C 180,E1 10258.442,E2 10258.442} C_VEL
LIN {X 0,Y 556.516,Z 859.31,A -85,B 0,C 180,E1 10263.123,E2 10263.123} C_VEL
LIN {X 0,Y 556.275,Z 859.31,A -85,B 0,C 180,E1 10267.828,E2 10267.828} C_VEL
LIN {X 0,Y 556.133,Z 859.31,A -85,B 0,C 180,E1 10272.589,E2 10272.589} C_VEL
LIN {X 0,Y 556.043,Z 859.31,A -85,B 0,C 180,E1 10277.484,E2 10277.484} C_VEL
LIN {X 0,Y 555.91,Z 859.31,A -85,B 0,C 180,E1 10282.429,E2 10282.429} C_VEL
LIN {X 0,Y 555.75,Z 859.31,A -85,B 0,C 180,E1 10287.609,E2 10287.609} C_VEL
LIN {X 0,Y 555.603,Z 859.31,A -85,B 0,C 180,E1 10293.049,E2 10293.049} C_VEL
LIN {X 0,Y 555.48,Z 859.31,A -85,B 0,C 180,E1 10298.85,E2 10298.85} C_VEL
LIN {X 0,Y 555.439,Z 859.31,A -85,B 0,C 180,E1 10304.821,E2 10304.821} C_VEL
LIN {X 0,Y 555.602,Z 860.104,A -85,B 0,C 180,E1 10308.999,E2 10308.999} C_VEL
LIN {X 0,Y 577.719,Z 906.946,A -85,B 0,C 180,E1 10311.424,E2 10311.424} C_VEL
LIN {X 0,Y 585.425,Z 927.82,A -85,B 0,C 180,E1 10312.336,E2 10312.336} C_VEL
LIN {X 0,Y 582.513,Z 974.365,A -85,B 0,C 180,E1 10313.513,E2 10313.513} C_VEL
LIN {X 0,Y 578.703,Z 1019.406,A -85,B 0,C 180,E1 10315.328,E2 10315.328} C_VEL
LIN {X 0,Y 574.692,Z 1056.395,A -85,B 0,C 180,E1 10317.379,E2 10317.379} C_VEL
LIN {X 0,Y 571.34,Z 1067.6,A -85,B 0,C 180,E1 10318,E2 10318} C_VEL
LIN {X 0,Y 564.508,Z 1083.737,A -85,B 0,C 180,E1 10318.924,E2 10318.924} C_VEL
LIN {X 0,Y 564.198,Z 1085.454,A -85,B 0,C 180,E1 10319.054,E2 10319.054} C_VEL
LIN {X 0,Y 559.769,Z 1119.946,A -85,B 0,C 180,E1 10322.111,E2 10322.111} C_VEL
LIN {X 0,Y 555.686,Z 1152.888,A -85,B 0,C 180,E1 10325.856,E2 10325.856} C_VEL
LIN {X 0,Y 552.662,Z 1180.773,A -85,B 0,C 180,E1 10329.957,E2 10329.957} C_VEL
LIN {X 0,Y 550.517,Z 1203.186,A -85,B 0,C 180,E1 10334.398,E2 10334.398} C_VEL
LIN {X 0,Y 549.399,Z 1219.145,A -85,B 0,C 180,E1 10338.868,E2 10338.868} C_VEL
LIN {X 0,Y 548.961,Z 1228.826,A -85,B 0,C 180,E1 10342.944,E2 10342.944} C_VEL
LIN {X 0,Y 548.779,Z 1233.849,A -85,B 0,C 180,E1 10346.834,E2 10346.834} C_VEL
LIN {X 0,Y 548.869,Z 1235.174,A -85,B 0,C 180,E1 10350,E2 10350} C_VEL
LIN {X 0,Y 548.869,Z 1232.236,A -85,B 0,C 180,E1 10354.751,E2 10354.751} C_VEL
LIN {X 0,Y 549.068,Z 1225.434,A -85,B 0,C 180,E1 10358.73,E2 10358.73} C_VEL
LIN {X 0,Y 549.797,Z 1212.703,A -85,B 0,C 180,E1 10363.143,E2 10363.143} C_VEL
LIN {X 0,Y 551.006,Z 1195.944,A -85,B 0,C 180,E1 10367.195,E2 10367.195} C_VEL
LIN {X 0,Y 553.435,Z 1172.049,A -85,B 0,C 180,E1 10371.455,E2 10371.455} C_VEL
LIN {X 0,Y 557.055,Z 1141.247,A -85,B 0,C 180,E1 10375.584,E2 10375.584} C_VEL
LIN {X 0,Y 561.85,Z 1104.399,A -85,B 0,C 180,E1 10379.368,E2 10379.368} C_VEL
LIN {X 0,Y 566.874,Z 1063.844,A -85,B 0,C 180,E1 10382.53,E2 10382.53} C_VEL
LIN {X 0,Y 571.787,Z 1020.469,A -85,B 0,C 180,E1 10385.035,E2 10385.035} C_VEL
LIN {X 0,Y 575.802,Z 976.534,A -85,B 0,C 180,E1 10386.834,E2 10386.834} C_VEL
LIN {X 0,Y 578.599,Z 931.947,A -85,B 0,C 180,E1 10388.026,E2 10388.026} C_VEL
LIN {X 0,Y 577.487,Z 925.985,A -85,B 0,C 180,E1 10388.245,E2 10388.245} C_VEL
LIN {X 0,Y 562.01,Z 888.82,A -85,B 0,C 180,E1 10390.018,E2 10390.018} C_VEL
LIN {X 0,Y 547.731,Z 860.263,A -85,B 0,C 180,E1 10391.642,E2 10391.642} C_VEL
LIN {X 0,Y 547.685,Z 859.31,A -85,B 0,C 180,E1 10391.681,E2 10391.681} C_VEL
LIN {X 0,Y 547.601,Z 859.31,A -85,B 0,C 180,E1 10396.24,E2 10396.24} C_VEL
LIN {X 0,Y 547.537,Z 859.31,A -85,B 0,C 180,E1 10402.503,E2 10402.503} C_VEL
LIN {X 0,Y 547.729,Z 859.31,A -85,B 0,C 180,E1 10408.296,E2 10408.296} C_VEL
LIN {X 0,Y 547.901,Z 859.31,A -85,B 0,C 180,E1 10413.742,E2 10413.742} C_VEL
LIN {X 0,Y 548.016,Z 859.31,A -85,B 0,C 180,E1 10418.937,E2 10418.937} C_VEL
LIN {X 0,Y 548.098,Z 859.31,A -85,B 0,C 180,E1 10423.953,E2 10423.953} C_VEL
LIN {X 0,Y 548.251,Z 859.31,A -85,B 0,C 180,E1 10428.845,E2 10428.845} C_VEL
LIN {X 0,Y 548.507,Z 859.31,A -85,B 0,C 180,E1 10434.002,E2 10434.002} C_VEL
LIN {X 0,Y 548.702,Z 859.31,A -85,B 0,C 180,E1 10439.998,E2 10439.998} C_VEL
LIN {X 0,Y 548.512,Z 859.31,A -85,B 0,C 180,E1 10446.004,E2 10446.004} C_VEL
LIN {X 0,Y 548.282,Z 859.31,A -85,B 0,C 180,E1 10451.15,E2 10451.15} C_VEL
LIN {X 0,Y 548.136,Z 859.31,A -85,B 0,C 180,E1 10456.041,E2 10456.041} C_VEL
LIN {X 0,Y 547.987,Z 859.31,A -85,B 0,C 180,E1 10461.06,E2 10461.06} C_VEL
LIN {X 0,Y 547.825,Z 859.31,A -85,B 0,C 180,E1 10466.258,E2 10466.258} C_VEL
LIN {X 0,Y 547.719,Z 859.31,A -85,B 0,C 180,E1 10471.7,E2 10471.7} C_VEL
LIN {X 0,Y 547.572,Z 859.31,A -85,B 0,C 180,E1 10477.489,E2 10477.489} C_VEL
LIN {X 0,Y 547.477,Z 859.31,A -85,B 0,C 180,E1 10483.767,E2 10483.767} C_VEL
LIN {X 0,Y 547.526,Z 859.31,A -85,B 0,C 180,E1 10488.379,E2 10488.379} C_VEL
LIN {X 0,Y 547.604,Z 859.31,A -85,B 0,C 180,E1 10493.342,E2 10493.342} C_VEL
LIN {X 0,Y 547.626,Z 859.602,A -85,B 0,C 180,E1 10494.542,E2 10494.542} C_VEL
LIN {X 0,Y 554.864,Z 874.167,A -85,B 0,C 180,E1 10495.351,E2 10495.351} C_VEL
LIN {X 0,Y 578.21,Z 921.112,A -85,B 0,C 180,E1 10497.772,E2 10497.772} C_VEL
LIN {X 0,Y 576.805,Z 972.924,A -85,B 0,C 180,E1 10498.561,E2 10498.561} C_VEL
LIN {X 0,Y 573.702,Z 1012.44,A -85,B 0,C 180,E1 10499.729,E2 10499.729} C_VEL
LIN {X 0,Y 569.515,Z 1050.726,A -85,B 0,C 180,E1 10501.516,E2 10501.516} C_VEL
LIN {X 0,Y 564.714,Z 1085.59,A -85,B 0,C 180,E1 10503.827,E2 10503.827} C_VEL
LIN {X 0,Y 560.079,Z 1116.068,A -85,B 0,C 180,E1 10506.564,E2 10506.564} C_VEL
LIN {X 0,Y 555.841,Z 1143.458,A -85,B 0,C 180,E1 10509.841,E2 10509.841} C_VEL
LIN {X 0,Y 552.56,Z 1166.47,A -85,B 0,C 180,E1 10513.538,E2 10513.538} C_VEL
LIN {X 0,Y 550.381,Z 1185.017,A -85,B 0,C 180,E1 10517.668,E2 10517.668} C_VEL
LIN {X 0,Y 549.41,Z 1196.313,A -85,B 0,C 180,E1 10521.275,E2 10521.275} C_VEL
LIN {X 0,Y 549.015,Z 1203.935,A -85,B 0,C 180,E1 10525.251,E2 10525.251} C_VEL
LIN {X 0,Y 548.813,Z 1206.782,A -85,B 0,C 180,E1 10528.418,E2 10528.418} C_VEL
LIN {X 0,Y 548.92,Z 1206.723,A -85,B 0,C 180,E1 10531.582,E2 10531.582} C_VEL
LIN {X 0,Y 549.096,Z 1202.657,A -85,B 0,C 180,E1 10535.543,E2 10535.543} C_VEL
LIN {X 0,Y 549.645,Z 1192.792,A -85,B 0,C 180,E1 10539.922,E2 10539.922} C_VEL
LIN {X 0,Y 551.08,Z 1178.308,A -85,B 0,C 180,E1 10543.922,E2 10543.922} C_VEL
LIN {X 0,Y 553.754,Z 1157.667,A -85,B 0,C 180,E1 10547.93,E2 10547.93} C_VEL
LIN {X 0,Y 557.604,Z 1132.266,A -85,B 0,C 180,E1 10551.523,E2 10551.523} C_VEL
LIN {X 0,Y 562.239,Z 1102.134,A -85,B 0,C 180,E1 10554.692,E2 10554.692} C_VEL
LIN {X 0,Y 567.035,Z 1069.578,A -85,B 0,C 180,E1 10557.235,E2 10557.235} C_VEL
LIN {X 0,Y 571.541,Z 1033.889,A -85,B 0,C 180,E1 10559.263,E2 10559.263} C_VEL
LIN {X 0,Y 575.184,Z 995.523,A -85,B 0,C 180,E1 10560.756,E2 10560.756} C_VEL
LIN {X 0,Y 577.464,Z 957.385,A -85,B 0,C 180,E1 10561.656,E2 10561.656} C_VEL
LIN {X 0,Y 577.591,Z 919.289,A -85,B 0,C 180,E1 10562.201,E2 10562.201} C_VEL
LIN {X 0,Y 549.654,Z 864.528,A -85,B 0,C 180,E1 10565.117,E2 10565.117} C_VEL
LIN {X 0,Y 547.648,Z 859.31,A -85,B 0,C 180,E1 10565.386,E2 10565.386} C_VEL
LIN {X 0,Y 547.612,Z 859.31,A -85,B 0,C 180,E1 10569.526,E2 10569.526} C_VEL
LIN {X 0,Y 547.474,Z 859.31,A -85,B 0,C 180,E1 10576.024,E2 10576.024} C_VEL
LIN {X 0,Y 547.577,Z 859.31,A -85,B 0,C 180,E1 10580.79,E2 10580.79} C_VEL
LIN {X 0,Y 547.636,Z 859.31,A -85,B 0,C 180,E1 10586.413,E2 10586.413} C_VEL
LIN {X 0,Y 547.797,Z 859.31,A -85,B 0,C 180,E1 10592.273,E2 10592.273} C_VEL
LIN {X 0,Y 547.929,Z 859.31,A -85,B 0,C 180,E1 10597.23,E2 10597.23} C_VEL
LIN {X 0,Y 547.887,Z 859.31,A -85,B 0,C 180,E1 10602.295,E2 10602.295} C_VEL
LIN {X 0,Y 548.153,Z 859.31,A -85,B 0,C 180,E1 10607.229,E2 10607.229} C_VEL
LIN {X 0,Y 548.479,Z 859.31,A -85,B 0,C 180,E1 10612.185,E2 10612.185} C_VEL
LIN {X 0,Y 548.647,Z 859.31,A -85,B 0,C 180,E1 10616.837,E2 10616.837} C_VEL
LIN {X 0,Y 548.766,Z 859.31,A -85,B 0,C 180,E1 10621.584,E2 10621.584} C_VEL
LIN {X 0,Y 548.506,Z 859.31,A -85,B 0,C 180,E1 10626.345,E2 10626.345} C_VEL
LIN {X 0,Y 548.268,Z 859.31,A -85,B 0,C 180,E1 10631.154,E2 10631.154} C_VEL
LIN {X 0,Y 548.14,Z 859.31,A -85,B 0,C 180,E1 10636.046,E2 10636.046} C_VEL
LIN {X 0,Y 548.019,Z 859.31,A -85,B 0,C 180,E1 10641.063,E2 10641.063} C_VEL
LIN {X 0,Y 547.863,Z 859.31,A -85,B 0,C 180,E1 10646.26,E2 10646.26} C_VEL
LIN {X 0,Y 547.736,Z 859.31,A -85,B 0,C 180,E1 10651.704,E2 10651.704} C_VEL
LIN {X 0,Y 547.553,Z 859.31,A -85,B 0,C 180,E1 10657.496,E2 10657.496} C_VEL
LIN {X 0,Y 547.475,Z 859.31,A -85,B 0,C 180,E1 10663.773,E2 10663.773} C_VEL
LIN {X 0,Y 547.58,Z 859.31,A -85,B 0,C 180,E1 10668.331,E2 10668.331} C_VEL
LIN {X 0,Y 554.174,Z 873.405,A -85,B 0,C 180,E1 10669.116,E2 10669.116} C_VEL
LIN {X 0,Y 572.241,Z 911.851,A -85,B 0,C 180,E1 10671.124,E2 10671.124} C_VEL
LIN {X 0,Y 578.788,Z 930.449,A -85,B 0,C 180,E1 10671.954,E2 10671.954} C_VEL
LIN {X 0,Y 575.78,Z 975.447,A -85,B 0,C 180,E1 10673.122,E2 10673.122} C_VEL
LIN {X 0,Y 571.914,Z 1018.953,A -85,B 0,C 180,E1 10674.894,E2 10674.894} C_VEL
LIN {X 0,Y 567.022,Z 1062.353,A -85,B 0,C 180,E1 10677.375,E2 10677.375} C_VEL
LIN {X 0,Y 564.198,Z 1085.454,A -85,B 0,C 180,E1 10679.054,E2 10679.054} C_VEL
LIN {X 0,Y 558.831,Z 1099.294,A -85,B 0,C 180,E1 10680.014,E2 10680.014} C_VEL
LIN {X 0,Y 553.434,Z 1112.563,A -85,B 0,C 180,E1 10681.051,E2 10681.051} C_VEL
LIN {X 0,Y 549.185,Z 1143.956,A -85,B 0,C 180,E1 10684.461,E2 10684.461} C_VEL
LIN {X 0,Y 545.592,Z 1173.144,A -85,B 0,C 180,E1 10688.524,E2 10688.524} C_VEL
LIN {X 0,Y 543.252,Z 1195.406,A -85,B 0,C 180,E1 10692.551,E2 10692.551} C_VEL
LIN {X 0,Y 541.918,Z 1212.315,A -85,B 0,C 180,E1 10696.662,E2 10696.662} C_VEL
LIN {X 0,Y 541.23,Z 1225.158,A -85,B 0,C 180,E1 10701.142,E2 10701.142} C_VEL
LIN {X 0,Y 540.985,Z 1232.017,A -85,B 0,C 180,E1 10705.18,E2 10705.18} C_VEL
LIN {X 0,Y 540.979,Z 1234.973,A -85,B 0,C 180,E1 10710,E2 10710} C_VEL
LIN {X 0,Y 540.992,Z 1232.016,A -85,B 0,C 180,E1 10714.82,E2 10714.82} C_VEL
LIN {X 0,Y 541.19,Z 1225.157,A -85,B 0,C 180,E1 10718.858,E2 10718.858} C_VEL
LIN {X 0,Y 541.96,Z 1212.299,A -85,B 0,C 180,E1 10723.336,E2 10723.336} C_VEL
LIN {X 0,Y 543.23,Z 1195.389,A -85,B 0,C 180,E1 10727.449,E2 10727.449} C_VEL
LIN {X 0,Y 545.796,Z 1171.333,A -85,B 0,C 180,E1 10731.771,E2 10731.771} C_VEL
LIN {X 0,Y 549.633,Z 1140.613,A -85,B 0,C 180,E1 10735.954,E2 10735.954} C_VEL
LIN {X 0,Y 554.664,Z 1104,A -85,B 0,C 180,E1 10739.758,E2 10739.758} C_VEL
LIN {X 0,Y 559.927,Z 1063.44,A -85,B 0,C 180,E1 10742.952,E2 10742.952} C_VEL
LIN {X 0,Y 565.053,Z 1020.064,A -85,B 0,C 180,E1 10745.478,E2 10745.478} C_VEL
LIN {X 0,Y 569.287,Z 975.658,A -85,B 0,C 180,E1 10747.305,E2 10747.305} C_VEL
LIN {X 0,Y 571.617,Z 930.294,A -85,B 0,C 180,E1 10748.549,E2 10748.549} C_VEL
LIN {X 0,Y 556.61,Z 893.592,A -85,B 0,C 180,E1 10750.351,E2 10750.351} C_VEL
LIN {X 0,Y 539.708,Z 859.763,A -85,B 0,C 180,E1 10752.328,E2 10752.328} C_VEL
LIN {X 0,Y 539.637,Z 859.31,A -85,B 0,C 180,E1 10757.641,E2 10757.641} C_VEL
LIN {X 0,Y 539.601,Z 859.31,A -85,B 0,C 180,E1 10763.872,E2 10763.872} C_VEL
LIN {X 0,Y 539.835,Z 859.31,A -85,B 0,C 180,E1 10769.658,E2 10769.658} C_VEL
LIN {X 0,Y 539.978,Z 859.31,A -85,B 0,C 180,E1 10775.111,E2 10775.111} C_VEL
LIN {X 0,Y 540.139,Z 859.31,A -85,B 0,C 180,E1 10780.331,E2 10780.331} C_VEL
LIN {X 0,Y 540.211,Z 859.31,A -85,B 0,C 180,E1 10785.379,E2 10785.379} C_VEL
LIN {X 0,Y 540.393,Z 859.31,A -85,B 0,C 180,E1 10790.315,E2 10790.315} C_VEL
LIN {X 0,Y 540.659,Z 859.31,A -85,B 0,C 180,E1 10795.176,E2 10795.176} C_VEL
LIN {X 0,Y 540.829,Z 859.31,A -85,B 0,C 180,E1 10799.998,E2 10799.998} C_VEL
LIN {X 0,Y 540.726,Z 859.31,A -85,B 0,C 180,E1 10804.819,E2 10804.819} C_VEL
LIN {X 0,Y 540.382,Z 859.31,A -85,B 0,C 180,E1 10811.315,E2 10811.315} C_VEL
LIN {X 0,Y 540.199,Z 859.31,A -85,B 0,C 180,E1 10817.5,E2 10817.5} C_VEL
LIN {X 0,Y 540.022,Z 859.31,A -85,B 0,C 180,E1 10823.122,E2 10823.122} C_VEL
LIN {X 0,Y 539.828,Z 859.31,A -85,B 0,C 180,E1 10828.491,E2 10828.491} C_VEL
LIN {X 0,Y 539.686,Z 859.31,A -85,B 0,C 180,E1 10834.15,E2 10834.15} C_VEL
LIN {X 0,Y 539.561,Z 859.31,A -85,B 0,C 180,E1 10840.219,E2 10840.219} C_VEL
LIN {X 0,Y 539.516,Z 859.31,A -85,B 0,C 180,E1 10845.4,E2 10845.4} C_VEL
LIN {X 0,Y 539.672,Z 859.31,A -85,B 0,C 180,E1 10851.807,E2 10851.807} C_VEL
LIN {X 0,Y 539.688,Z 859.31,A -85,B 0,C 180,E1 10853.834,E2 10853.834} C_VEL
LIN {X 0,Y 544.495,Z 869.589,A -85,B 0,C 180,E1 10854.426,E2 10854.426} C_VEL
LIN {X 0,Y 571.776,Z 923.144,A -85,B 0,C 180,E1 10857.336,E2 10857.336} C_VEL
LIN {X 0,Y 570.36,Z 972.451,A -85,B 0,C 180,E1 10858.098,E2 10858.098} C_VEL
LIN {X 0,Y 567.209,Z 1011.36,A -85,B 0,C 180,E1 10859.245,E2 10859.245} C_VEL
LIN {X 0,Y 562.854,Z 1049.473,A -85,B 0,C 180,E1 10861.015,E2 10861.015} C_VEL
LIN {X 0,Y 557.812,Z 1085.109,A -85,B 0,C 180,E1 10863.385,E2 10863.385} C_VEL
LIN {X 0,Y 552.791,Z 1116.566,A -85,B 0,C 180,E1 10866.241,E2 10866.241} C_VEL
LIN {X 0,Y 548.389,Z 1143.541,A -85,B 0,C 180,E1 10869.511,E2 10869.511} C_VEL
LIN {X 0,Y 544.933,Z 1166.49,A -85,B 0,C 180,E1 10873.239,E2 10873.239} C_VEL
LIN {X 0,Y 542.757,Z 1183.88,A -85,B 0,C 180,E1 10877.094,E2 10877.094} C_VEL
LIN {X 0,Y 541.561,Z 1196.56,A -85,B 0,C 180,E1 10881.148,E2 10881.148} C_VEL
LIN {X 0,Y 541.126,Z 1204.152,A -85,B 0,C 180,E1 10885.181,E2 10885.181} C_VEL
LIN {X 0,Y 540.936,Z 1206.985,A -85,B 0,C 180,E1 10888.395,E2 10888.395} C_VEL
LIN {X 0,Y 541.035,Z 1206.927,A -85,B 0,C 180,E1 10891.605,E2 10891.605} C_VEL
LIN {X 0,Y 541.226,Z 1202.877,A -85,B 0,C 180,E1 10895.624,E2 10895.624} C_VEL
LIN {X 0,Y 541.829,Z 1193.045,A -85,B 0,C 180,E1 10900.067,E2 10900.067} C_VEL
LIN {X 0,Y 543.557,Z 1176.832,A -85,B 0,C 180,E1 10904.531,E2 10904.531} C_VEL
LIN {X 0,Y 546.522,Z 1155.492,A -85,B 0,C 180,E1 10908.594,E2 10908.594} C_VEL
LIN {X 0,Y 550.47,Z 1131.012,A -85,B 0,C 180,E1 10912.028,E2 10912.028} C_VEL
LIN {X 0,Y 555.206,Z 1101.558,A -85,B 0,C 180,E1 10915.134,E2 10915.134} C_VEL
LIN {X 0,Y 560.204,Z 1068.893,A -85,B 0,C 180,E1 10917.696,E2 10917.696} C_VEL
LIN {X 0,Y 564.973,Z 1032.742,A -85,B 0,C 180,E1 10919.748,E2 10919.748} C_VEL
LIN {X 0,Y 568.667,Z 994.923,A -85,B 0,C 180,E1 10921.222,E2 10921.222} C_VEL
LIN {X 0,Y 571.087,Z 955.497,A -85,B 0,C 180,E1 10922.141,E2 10922.141} C_VEL
LIN {X 0,Y 571.118,Z 921.795,A -85,B 0,C 180,E1 10922.635,E2 10922.635} C_VEL
LIN {X 0,Y 544.674,Z 869.806,A -85,B 0,C 180,E1 10925.456,E2 10925.456} C_VEL
LIN {X 0,Y 539.683,Z 859.31,A -85,B 0,C 180,E1 10926.131,E2 10926.131} C_VEL
LIN {X 0,Y 539.549,Z 859.31,A -85,B 0,C 180,E1 10932.379,E2 10932.379} C_VEL
LIN {X 0,Y 539.543,Z 859.31,A -85,B 0,C 180,E1 10937.638,E2 10937.638} C_VEL
LIN {X 0,Y 539.66,Z 859.31,A -85,B 0,C 180,E1 10943.882,E2 10943.882} C_VEL
LIN {X 0,Y 539.808,Z 859.31,A -85,B 0,C 180,E1 10949.662,E2 10949.662} C_VEL
LIN {X 0,Y 539.934,Z 859.31,A -85,B 0,C 180,E1 10955.114,E2 10955.114} C_VEL
LIN {X 0,Y 539.993,Z 859.31,A -85,B 0,C 180,E1 10960.33,E2 10960.33} C_VEL
LIN {X 0,Y 540.214,Z 859.31,A -85,B 0,C 180,E1 10967.038,E2 10967.038} C_VEL
LIN {X 0,Y 540.546,Z 859.31,A -85,B 0,C 180,E1 10972.179,E2 10972.179} C_VEL
LIN {X 0,Y 540.739,Z 859.31,A -85,B 0,C 180,E1 10976.79,E2 10976.79} C_VEL
LIN {X 0,Y 540.863,Z 859.31,A -85,B 0,C 180,E1 10981.607,E2 10981.607} C_VEL
LIN {X 0,Y 540.585,Z 859.31,A -85,B 0,C 180,E1 10986.438,E2 10986.438} C_VEL
LIN {X 0,Y 540.356,Z 859.31,A -85,B 0,C 180,E1 10991.32,E2 10991.32} C_VEL
LIN {X 0,Y 540.231,Z 859.31,A -85,B 0,C 180,E1 10997.509,E2 10997.509} C_VEL
LIN {X 0,Y 540.045,Z 859.31,A -85,B 0,C 180,E1 11003.126,E2 11003.126} C_VEL
LIN {X 0,Y 539.852,Z 859.31,A -85,B 0,C 180,E1 11008.495,E2 11008.495} C_VEL
LIN {X 0,Y 539.688,Z 859.31,A -85,B 0,C 180,E1 11014.155,E2 11014.155} C_VEL
LIN {X 0,Y 539.562,Z 859.31,A -85,B 0,C 180,E1 11020.225,E2 11020.225} C_VEL
LIN {X 0,Y 539.516,Z 859.31,A -85,B 0,C 180,E1 11025.4,E2 11025.4} C_VEL
LIN {X 0,Y 539.578,Z 859.414,A -85,B 0,C 180,E1 11027.662,E2 11027.662} C_VEL
LIN {X 0,Y 544.509,Z 869.791,A -85,B 0,C 180,E1 11028.266,E2 11028.266} C_VEL
LIN {X 0,Y 564.899,Z 912.072,A -85,B 0,C 180,E1 11030.597,E2 11030.597} C_VEL
LIN {X 0,Y 572.163,Z 933.085,A -85,B 0,C 180,E1 11031.561,E2 11031.561} C_VEL
LIN {X 0,Y 569.124,Z 975.716,A -85,B 0,C 180,E1 11032.69,E2 11032.69} C_VEL
LIN {X 0,Y 565.031,Z 1019.986,A -85,B 0,C 180,E1 11034.519,E2 11034.519} C_VEL
LIN {X 0,Y 559.883,Z 1063.536,A -85,B 0,C 180,E1 11037.055,E2 11037.055} C_VEL
LIN {X 0,Y 554.619,Z 1103.973,A -85,B 0,C 180,E1 11040.239,E2 11040.239} C_VEL
LIN {X 0,Y 553.434,Z 1112.563,A -85,B 0,C 180,E1 11041.051,E2 11041.051} C_VEL
LIN {X 0,Y 548.017,Z 1125.336,A -85,B 0,C 180,E1 11042.173,E2 11042.173} C_VEL
LIN {X 0,Y 542.652,Z 1137.49,A -85,B 0,C 180,E1 11043.371,E2 11043.371} C_VEL
LIN {X 0,Y 538.752,Z 1166.371,A -85,B 0,C 180,E1 11047.24,E2 11047.24} C_VEL
LIN {X 0,Y 535.945,Z 1190.583,A -85,B 0,C 180,E1 11051.423,E2 11051.423} C_VEL
LIN {X 0,Y 534.253,Z 1208.951,A -85,B 0,C 180,E1 11055.63,E2 11055.63} C_VEL
LIN {X 0,Y 533.415,Z 1222.869,A -85,B 0,C 180,E1 11060.186,E2 11060.186} C_VEL
LIN {X 0,Y 533.167,Z 1230.286,A -85,B 0,C 180,E1 11063.986,E2 11063.986} C_VEL
LIN {X 0,Y 533.109,Z 1234.425,A -85,B 0,C 180,E1 11068.371,E2 11068.371} C_VEL
LIN {X 0,Y 533.079,Z 1233.431,A -85,B 0,C 180,E1 11073.259,E2 11073.259} C_VEL
LIN {X 0,Y 533.145,Z 1228.144,A -85,B 0,C 180,E1 11077.348,E2 11077.348} C_VEL
LIN {X 0,Y 533.759,Z 1217.039,A -85,B 0,C 180,E1 11081.954,E2 11081.954} C_VEL
LIN {X 0,Y 535.045,Z 1200.517,A -85,B 0,C 180,E1 11086.452,E2 11086.452} C_VEL
LIN {X 0,Y 537.352,Z 1178.208,A -85,B 0,C 180,E1 11090.855,E2 11090.855} C_VEL
LIN {X 0,Y 540.967,Z 1150.09,A -85,B 0,C 180,E1 11095.066,E2 11095.066} C_VEL
LIN {X 0,Y 545.676,Z 1116.063,A -85,B 0,C 180,E1 11098.971,E2 11098.971} C_VEL
LIN {X 0,Y 551.012,Z 1077.952,A -85,B 0,C 180,E1 11102.312,E2 11102.312} C_VEL
LIN {X 0,Y 556.556,Z 1034.938,A -85,B 0,C 180,E1 11105.131,E2 11105.131} C_VEL
LIN {X 0,Y 561.321,Z 990.31,A -85,B 0,C 180,E1 11107.234,E2 11107.234} C_VEL
LIN {X 0,Y 565.075,Z 942.691,A -85,B 0,C 180,E1 11108.706,E2 11108.706} C_VEL
LIN {X 0,Y 565.027,Z 932.642,A -85,B 0,C 180,E1 11108.963,E2 11108.963} C_VEL
LIN {X 0,Y 550.958,Z 897.791,A -85,B 0,C 180,E1 11110.722,E2 11110.722} C_VEL
LIN {X 0,Y 531.808,Z 859.761,A -85,B 0,C 180,E1 11113.023,E2 11113.023} C_VEL
LIN {X 0,Y 531.694,Z 859.31,A -85,B 0,C 180,E1 11119.054,E2 11119.054} C_VEL
LIN {X 0,Y 531.708,Z 859.31,A -85,B 0,C 180,E1 11125.26,E2 11125.26} C_VEL
LIN {X 0,Y 531.937,Z 859.31,A -85,B 0,C 180,E1 11131.041,E2 11131.041} C_VEL
LIN {X 0,Y 532.102,Z 859.31,A -85,B 0,C 180,E1 11136.508,E2 11136.508} C_VEL
LIN {X 0,Y 532.271,Z 859.31,A -85,B 0,C 180,E1 11141.753,E2 11141.753} C_VEL
LIN {X 0,Y 532.314,Z 859.31,A -85,B 0,C 180,E1 11146.838,E2 11146.838} C_VEL
LIN {X 0,Y 532.617,Z 859.31,A -85,B 0,C 180,E1 11151.822,E2 11151.822} C_VEL
LIN {X 0,Y 532.826,Z 859.31,A -85,B 0,C 180,E1 11156.738,E2 11156.738} C_VEL
LIN {X 0,Y 532.951,Z 859.31,A -85,B 0,C 180,E1 11161.627,E2 11161.627} C_VEL
LIN {X 0,Y 532.672,Z 859.31,A -85,B 0,C 180,E1 11166.53,E2 11166.53} C_VEL
LIN {X 0,Y 532.454,Z 859.31,A -85,B 0,C 180,E1 11171.485,E2 11171.485} C_VEL
LIN {X 0,Y 532.312,Z 859.31,A -85,B 0,C 180,E1 11176.532,E2 11176.532} C_VEL
LIN {X 0,Y 532.133,Z 859.31,A -85,B 0,C 180,E1 11181.719,E2 11181.719} C_VEL
LIN {X 0,Y 531.894,Z 859.31,A -85,B 0,C 180,E1 11187.976,E2 11187.976} C_VEL
LIN {X 0,Y 531.773,Z 859.31,A -85,B 0,C 180,E1 11194.274,E2 11194.274} C_VEL
LIN {X 0,Y 531.608,Z 859.31,A -85,B 0,C 180,E1 11199.682,E2 11199.682} C_VEL
LIN {X 0,Y 531.614,Z 859.31,A -85,B 0,C 180,E1 11205.427,E2 11205.427} C_VEL
LIN {X 0,Y 531.698,Z 859.31,A -85,B 0,C 180,E1 11211.173,E2 11211.173} C_VEL
LIN {X 0,Y 531.824,Z 859.31,A -85,B 0,C 180,E1 11213.122,E2 11213.122} C_VEL
LIN {X 0,Y 536.899,Z 870.06,A -85,B 0,C 180,E1 11213.776,E2 11213.776} C_VEL
LIN {X 0,Y 562.171,Z 919.278,A -85,B 0,C 180,E1 11216.566,E2 11216.566} C_VEL
LIN {X 0,Y 565.324,Z 927.732,A -85,B 0,C 180,E1 11216.922,E2 11216.922} C_VEL
LIN {X 0,Y 563.856,Z 973.229,A -85,B 0,C 180,E1 11217.654,E2 11217.654} C_VEL
LIN {X 0,Y 560.537,Z 1012.214,A -85,B 0,C 180,E1 11218.827,E2 11218.827} C_VEL
LIN {X 0,Y 555.979,Z 1050.216,A -85,B 0,C 180,E1 11220.621,E2 11220.621} C_VEL
LIN {X 0,Y 550.77,Z 1085.498,A -85,B 0,C 180,E1 11223.003,E2 11223.003} C_VEL
LIN {X 0,Y 545.763,Z 1115.948,A -85,B 0,C 180,E1 11225.792,E2 11225.792} C_VEL
LIN {X 0,Y 540.87,Z 1144.09,A -85,B 0,C 180,E1 11229.241,E2 11229.241} C_VEL
LIN {X 0,Y 537.288,Z 1166.763,A -85,B 0,C 180,E1 11232.986,E2 11232.986} C_VEL
LIN {X 0,Y 534.821,Z 1185.375,A -85,B 0,C 180,E1 11237.25,E2 11237.25} C_VEL
LIN {X 0,Y 533.714,Z 1196.799,A -85,B 0,C 180,E1 11241.017,E2 11241.017} C_VEL
LIN {X 0,Y 533.236,Z 1204.366,A -85,B 0,C 180,E1 11245.11,E2 11245.11} C_VEL
LIN {X 0,Y 533.038,Z 1207.189,A -85,B 0,C 180,E1 11248.371,E2 11248.371} C_VEL
LIN {X 0,Y 533.135,Z 1207.131,A -85,B 0,C 180,E1 11251.629,E2 11251.629} C_VEL
LIN {X 0,Y 533.346,Z 1202.232,A -85,B 0,C 180,E1 11256.235,E2 11256.235} C_VEL
LIN {X 0,Y 534.12,Z 1192.066,A -85,B 0,C 180,E1 11260.627,E2 11260.627} C_VEL
LIN {X 0,Y 535.831,Z 1177.13,A -85,B 0,C 180,E1 11264.745,E2 11264.745} C_VEL
LIN {X 0,Y 538.949,Z 1155.843,A -85,B 0,C 180,E1 11268.865,E2 11268.865} C_VEL
LIN {X 0,Y 543.326,Z 1129.743,A -85,B 0,C 180,E1 11272.549,E2 11272.549} C_VEL
LIN {X 0,Y 548.235,Z 1100.959,A -85,B 0,C 180,E1 11275.586,E2 11275.586} C_VEL
LIN {X 0,Y 553.44,Z 1068.071,A -85,B 0,C 180,E1 11278.176,E2 11278.176} C_VEL
LIN {X 0,Y 558.273,Z 1032.654,A -85,B 0,C 180,E1 11280.198,E2 11280.198} C_VEL
LIN {X 0,Y 562.164,Z 994.612,A -85,B 0,C 180,E1 11281.688,E2 11281.688} C_VEL
LIN {X 0,Y 564.721,Z 954.143,A -85,B 0,C 180,E1 11282.627,E2 11282.627} C_VEL
LIN {X 0,Y 564.66,Z 924.387,A -85,B 0,C 180,E1 11283.078,E2 11283.078} C_VEL
LIN {X 0,Y 539.312,Z 874.461,A -85,B 0,C 180,E1 11285.845,E2 11285.845} C_VEL
LIN {X 0,Y 531.835,Z 860.595,A -85,B 0,C 180,E1 11286.721,E2 11286.721} C_VEL
LIN {X 0,Y 531.709,Z 859.31,A -85,B 0,C 180,E1 11286.761,E2 11286.761} C_VEL
LIN {X 0,Y 531.642,Z 859.31,A -85,B 0,C 180,E1 11292.199,E2 11292.199} C_VEL
LIN {X 0,Y 531.634,Z 859.31,A -85,B 0,C 180,E1 11297.823,E2 11297.823} C_VEL
LIN {X 0,Y 531.679,Z 859.31,A -85,B 0,C 180,E1 11303.251,E2 11303.251} C_VEL
LIN {X 0,Y 531.833,Z 859.31,A -85,B 0,C 180,E1 11309.158,E2 11309.158} C_VEL
LIN {X 0,Y 532.01,Z 859.31,A -85,B 0,C 180,E1 11314.717,E2 11314.717} C_VEL
LIN {X 0,Y 532.06,Z 859.31,A -85,B 0,C 180,E1 11320.024,E2 11320.024} C_VEL
LIN {X 0,Y 532.201,Z 859.31,A -85,B 0,C 180,E1 11325.479,E2 11325.479} C_VEL
LIN {X 0,Y 532.508,Z 859.31,A -85,B 0,C 180,E1 11330.174,E2 11330.174} C_VEL
LIN {X 0,Y 532.758,Z 859.31,A -85,B 0,C 180,E1 11335.109,E2 11335.109} C_VEL
LIN {X 0,Y 532.936,Z 859.31,A -85,B 0,C 180,E1 11340.002,E2 11340.002} C_VEL
LIN {X 0,Y 532.731,Z 859.31,A -85,B 0,C 180,E1 11345.413,E2 11345.413} C_VEL
LIN {X 0,Y 532.427,Z 859.31,A -85,B 0,C 180,E1 11351.491,E2 11351.491} C_VEL
LIN {X 0,Y 532.324,Z 859.31,A -85,B 0,C 180,E1 11356.536,E2 11356.536} C_VEL
LIN {X 0,Y 532.171,Z 859.31,A -85,B 0,C 180,E1 11361.722,E2 11361.722} C_VEL
LIN {X 0,Y 531.922,Z 859.31,A -85,B 0,C 180,E1 11367.981,E2 11367.981} C_VEL
LIN {X 0,Y 531.773,Z 859.31,A -85,B 0,C 180,E1 11374.273,E2 11374.273} C_VEL
LIN {X 0,Y 531.608,Z 859.31,A -85,B 0,C 180,E1 11379.681,E2 11379.681} C_VEL
LIN {X 0,Y 531.613,Z 859.31,A -85,B 0,C 180,E1 11385.434,E2 11385.434} C_VEL
LIN {X 0,Y 531.665,Z 859.602,A -85,B 0,C 180,E1 11386.97,E2 11386.97} C_VEL
LIN {X 0,Y 541.469,Z 878.968,A -85,B 0,C 180,E1 11388.176,E2 11388.176} C_VEL
LIN {X 0,Y 560.035,Z 918.65,A -85,B 0,C 180,E1 11390.364,E2 11390.364} C_VEL
LIN {X 0,Y 565.552,Z 935.709,A -85,B 0,C 180,E1 11391.156,E2 11391.156} C_VEL
LIN {X 0,Y 562.341,Z 978.114,A -85,B 0,C 180,E1 11392.324,E2 11392.324} C_VEL
LIN {X 0,Y 558.131,Z 1021.463,A -85,B 0,C 180,E1 11394.159,E2 11394.159} C_VEL
LIN {X 0,Y 552.717,Z 1065.011,A -85,B 0,C 180,E1 11396.749,E2 11396.749} C_VEL
LIN {X 0,Y 547.3,Z 1104.652,A -85,B 0,C 180,E1 11399.933,E2 11399.933} C_VEL
LIN {X 0,Y 542.652,Z 1137.49,A -85,B 0,C 180,E1 11403.371,E2 11403.371} C_VEL
LIN {X 0,Y 537.26,Z 1149.088,A -85,B 0,C 180,E1 11404.651,E2 11404.651} C_VEL
LIN {X 0,Y 532.054,Z 1160.015,A -85,B 0,C 180,E1 11406.009,E2 11406.009} C_VEL
LIN {X 0,Y 528.756,Z 1185.506,A -85,B 0,C 180,E1 11410.243,E2 11410.243} C_VEL
LIN {X 0,Y 526.777,Z 1205.364,A -85,B 0,C 180,E1 11414.59,E2 11414.59} C_VEL
LIN {X 0,Y 525.7,Z 1220.592,A -85,B 0,C 180,E1 11419.23,E2 11419.23} C_VEL
LIN {X 0,Y 525.268,Z 1230.167,A -85,B 0,C 180,E1 11423.976,E2 11423.976} C_VEL
LIN {X 0,Y 525.226,Z 1234.222,A -85,B 0,C 180,E1 11428.347,E2 11428.347} C_VEL
LIN {X 0,Y 525.123,Z 1234.219,A -85,B 0,C 180,E1 11431.653,E2 11431.653} C_VEL
LIN {X 0,Y 525.27,Z 1229.243,A -85,B 0,C 180,E1 11436.626,E2 11436.626} C_VEL
LIN {X 0,Y 525.742,Z 1219.441,A -85,B 0,C 180,E1 11441.174,E2 11441.174} C_VEL
LIN {X 0,Y 526.917,Z 1203.805,A -85,B 0,C 180,E1 11445.818,E2 11445.818} C_VEL
LIN {X 0,Y 529.423,Z 1180.23,A -85,B 0,C 180,E1 11450.744,E2 11450.744} C_VEL
LIN {X 0,Y 533.307,Z 1151.213,A -85,B 0,C 180,E1 11455.226,E2 11455.226} C_VEL
LIN {X 0,Y 538.293,Z 1116.882,A -85,B 0,C 180,E1 11459.255,E2 11459.255} C_VEL
LIN {X 0,Y 544.01,Z 1077.914,A -85,B 0,C 180,E1 11462.724,E2 11462.724} C_VEL
LIN {X 0,Y 549.772,Z 1035.073,A -85,B 0,C 180,E1 11465.564,E2 11465.564} C_VEL
LIN {X 0,Y 554.772,Z 990.05,A -85,B 0,C 180,E1 11467.704,E2 11467.704} C_VEL
LIN {X 0,Y 558.641,Z 942.519,A -85,B 0,C 180,E1 11469.182,E2 11469.182} C_VEL
LIN {X 0,Y 558.188,Z 934.054,A -85,B 0,C 180,E1 11469.432,E2 11469.432} C_VEL
LIN {X 0,Y 545.019,Z 901.282,A -85,B 0,C 180,E1 11471.139,E2 11471.139} C_VEL
LIN {X 0,Y 523.88,Z 860.115,A -85,B 0,C 180,E1 11473.742,E2 11473.742} C_VEL
LIN {X 0,Y 523.794,Z 859.31,A -85,B 0,C 180,E1 11478.777,E2 11478.777} C_VEL
LIN {X 0,Y 523.716,Z 859.31,A -85,B 0,C 180,E1 11484.651,E2 11484.651} C_VEL
LIN {X 0,Y 523.96,Z 859.31,A -85,B 0,C 180,E1 11490.558,E2 11490.558} C_VEL
LIN {X 0,Y 524.179,Z 859.31,A -85,B 0,C 180,E1 11496.131,E2 11496.131} C_VEL
LIN {X 0,Y 524.324,Z 859.31,A -85,B 0,C 180,E1 11501.467,E2 11501.467} C_VEL
LIN {X 0,Y 524.399,Z 859.31,A -85,B 0,C 180,E1 11506.636,E2 11506.636} C_VEL
LIN {X 0,Y 524.69,Z 859.31,A -85,B 0,C 180,E1 11511.697,E2 11511.697} C_VEL
LIN {X 0,Y 524.932,Z 859.31,A -85,B 0,C 180,E1 11516.689,E2 11516.689} C_VEL
LIN {X 0,Y 525.044,Z 859.31,A -85,B 0,C 180,E1 11521.651,E2 11521.651} C_VEL
LIN {X 0,Y 524.754,Z 859.31,A -85,B 0,C 180,E1 11526.629,E2 11526.629} C_VEL
LIN {X 0,Y 524.536,Z 859.31,A -85,B 0,C 180,E1 11531.661,E2 11531.661} C_VEL
LIN {X 0,Y 524.34,Z 859.31,A -85,B 0,C 180,E1 11537.51,E2 11537.51} C_VEL
LIN {X 0,Y 524.163,Z 859.31,A -85,B 0,C 180,E1 11542.32,E2 11542.32} C_VEL
LIN {X 0,Y 524.018,Z 859.31,A -85,B 0,C 180,E1 11547.549,E2 11547.549} C_VEL
LIN {X 0,Y 523.861,Z 859.31,A -85,B 0,C 180,E1 11553.326,E2 11553.326} C_VEL
LIN {X 0,Y 523.707,Z 859.31,A -85,B 0,C 180,E1 11559.519,E2 11559.519} C_VEL
LIN {X 0,Y 523.697,Z 859.31,A -85,B 0,C 180,E1 11566.019,E2 11566.019} C_VEL
LIN {X 0,Y 523.838,Z 859.31,A -85,B 0,C 180,E1 11572.398,E2 11572.398} C_VEL
LIN {X 0,Y 528.458,Z 869.213,A -85,B 0,C 180,E1 11573.004,E2 11573.004} C_VEL
LIN {X 0,Y 552.836,Z 915.553,A -85,B 0,C 180,E1 11575.786,E2 11575.786} C_VEL
LIN {X 0,Y 558.96,Z 929.907,A -85,B 0,C 180,E1 11576.469,E2 11576.469} C_VEL
LIN {X 0,Y 557.347,Z 974.448,A -85,B 0,C 180,E1 11577.211,E2 11577.211} C_VEL
LIN {X 0,Y 553.946,Z 1012.691,A -85,B 0,C 180,E1 11578.386,E2 11578.386} C_VEL
LIN {X 0,Y 549.137,Z 1050.941,A -85,B 0,C 180,E1 11580.219,E2 11580.219} C_VEL
LIN {X 0,Y 543.786,Z 1085.668,A -85,B 0,C 180,E1 11582.593,E2 11582.593} C_VEL
LIN {X 0,Y 538.444,Z 1116.657,A -85,B 0,C 180,E1 11585.475,E2 11585.475} C_VEL
LIN {X 0,Y 533.565,Z 1143.617,A -85,B 0,C 180,E1 11588.815,E2 11588.815} C_VEL
LIN {X 0,Y 529.637,Z 1167.062,A -85,B 0,C 180,E1 11592.733,E2 11592.733} C_VEL
LIN {X 0,Y 527.176,Z 1184.407,A -85,B 0,C 180,E1 11596.706,E2 11596.706} C_VEL
LIN {X 0,Y 525.852,Z 1197.032,A -85,B 0,C 180,E1 11600.881,E2 11600.881} C_VEL
LIN {X 0,Y 525.371,Z 1204.577,A -85,B 0,C 180,E1 11605.036,E2 11605.036} C_VEL
LIN {X 0,Y 525.176,Z 1207.725,A -85,B 0,C 180,E1 11610,E2 11610} C_VEL
LIN {X 0,Y 525.227,Z 1206.248,A -85,B 0,C 180,E1 11613.308,E2 11613.308} C_VEL
LIN {X 0,Y 525.618,Z 1200.451,A -85,B 0,C 180,E1 11617.454,E2 11617.454} C_VEL
LIN {X 0,Y 526.751,Z 1188.237,A -85,B 0,C 180,E1 11622.104,E2 11622.104} C_VEL
LIN {X 0,Y 528.998,Z 1170.775,A -85,B 0,C 180,E1 11626.431,E2 11626.431} C_VEL
LIN {X 0,Y 532.683,Z 1148.63,A -85,B 0,C 180,E1 11630.35,E2 11630.35} C_VEL
LIN {X 0,Y 537.528,Z 1121.462,A -85,B 0,C 180,E1 11633.903,E2 11633.903} C_VEL
LIN {X 0,Y 542.792,Z 1091.583,A -85,B 0,C 180,E1 11636.826,E2 11636.826} C_VEL
LIN {X 0,Y 548.317,Z 1056.582,A -85,B 0,C 180,E1 11639.352,E2 11639.352} C_VEL
LIN {X 0,Y 553.179,Z 1019.413,A -85,B 0,C 180,E1 11641.248,E2 11641.248} C_VEL
LIN {X 0,Y 556.759,Z 981.066,A -85,B 0,C 180,E1 11642.542,E2 11642.542} C_VEL
LIN {X 0,Y 558.708,Z 938.992,A -85,B 0,C 180,E1 11643.325,E2 11643.325} C_VEL
LIN {X 0,Y 558.22,Z 926.854,A -85,B 0,C 180,E1 11643.533,E2 11643.533} C_VEL
LIN {X 0,Y 533.73,Z 878.593,A -85,B 0,C 180,E1 11646.272,E2 11646.272} C_VEL
LIN {X 0,Y 523.806,Z 860.021,A -85,B 0,C 180,E1 11647.472,E2 11647.472} C_VEL
LIN {X 0,Y 523.737,Z 859.31,A -85,B 0,C 180,E1 11651.717,E2 11651.717} C_VEL
LIN {X 0,Y 523.727,Z 859.31,A -85,B 0,C 180,E1 11658.299,E2 11658.299} C_VEL
LIN {X 0,Y 523.788,Z 859.31,A -85,B 0,C 180,E1 11664.662,E2 11664.662} C_VEL
LIN {X 0,Y 523.918,Z 859.31,A -85,B 0,C 180,E1 11670.56,E2 11670.56} C_VEL
LIN {X 0,Y 524.144,Z 859.31,A -85,B 0,C 180,E1 11676.135,E2 11676.135} C_VEL
LIN {X 0,Y 524.123,Z 859.31,A -85,B 0,C 180,E1 11681.464,E2 11681.464} C_VEL
LIN {X 0,Y 524.352,Z 859.31,A -85,B 0,C 180,E1 11686.639,E2 11686.639} C_VEL
LIN {X 0,Y 524.701,Z 859.31,A -85,B 0,C 180,E1 11692.171,E2 11692.171} C_VEL
LIN {X 0,Y 524.936,Z 859.31,A -85,B 0,C 180,E1 11696.693,E2 11696.693} C_VEL
LIN {X 0,Y 525.049,Z 859.31,A -85,B 0,C 180,E1 11701.656,E2 11701.656} C_VEL
LIN {X 0,Y 524.745,Z 859.31,A -85,B 0,C 180,E1 11706.633,E2 11706.633} C_VEL
LIN {X 0,Y 524.516,Z 859.31,A -85,B 0,C 180,E1 11711.666,E2 11711.666} C_VEL
LIN {X 0,Y 524.343,Z 859.31,A -85,B 0,C 180,E1 11717.51,E2 11717.51} C_VEL
LIN {X 0,Y 524.197,Z 859.31,A -85,B 0,C 180,E1 11722.328,E2 11722.328} C_VEL
LIN {X 0,Y 524.049,Z 859.31,A -85,B 0,C 180,E1 11727.552,E2 11727.552} C_VEL
LIN {X 0,Y 523.871,Z 859.31,A -85,B 0,C 180,E1 11733.33,E2 11733.33} C_VEL
LIN {X 0,Y 523.708,Z 859.31,A -85,B 0,C 180,E1 11739.525,E2 11739.525} C_VEL
LIN {X 0,Y 523.688,Z 859.31,A -85,B 0,C 180,E1 11746.017,E2 11746.017} C_VEL
LIN {X 0,Y 523.71,Z 859.31,A -85,B 0,C 180,E1 11746.229,E2 11746.229} C_VEL
LIN {X 0,Y 527.993,Z 868.898,A -85,B 0,C 180,E1 11746.813,E2 11746.813} C_VEL
LIN {X 0,Y 549.425,Z 910.744,A -85,B 0,C 180,E1 11749.388,E2 11749.388} C_VEL
LIN {X 0,Y 559.018,Z 938.057,A -85,B 0,C 180,E1 11750.737,E2 11750.737} C_VEL
LIN {X 0,Y 555.496,Z 981.423,A -85,B 0,C 180,E1 11751.981,E2 11751.981} C_VEL
LIN {X 0,Y 551.286,Z 1022.634,A -85,B 0,C 180,E1 11753.775,E2 11753.775} C_VEL
LIN {X 0,Y 545.889,Z 1064.304,A -85,B 0,C 180,E1 11756.278,E2 11756.278} C_VEL
LIN {X 0,Y 540.145,Z 1104.26,A -85,B 0,C 180,E1 11759.513,E2 11759.513} C_VEL
LIN {X 0,Y 534.937,Z 1139.523,A -85,B 0,C 180,E1 11763.276,E2 11763.276} C_VEL
LIN {X 0,Y 532.054,Z 1160.015,A -85,B 0,C 180,E1 11766.009,E2 11766.009} C_VEL
LIN {X 0,Y 526.864,Z 1170.381,A -85,B 0,C 180,E1 11767.434,E2 11767.434} C_VEL
LIN {X 0,Y 521.771,Z 1179.869,A -85,B 0,C 180,E1 11768.95,E2 11768.95} C_VEL
LIN {X 0,Y 519.144,Z 1202.922,A -85,B 0,C 180,E1 11773.81,E2 11773.81} C_VEL
LIN {X 0,Y 517.865,Z 1219.125,A -85,B 0,C 180,E1 11778.662,E2 11778.662} C_VEL
LIN {X 0,Y 517.395,Z 1229.001,A -85,B 0,C 180,E1 11783.272,E2 11783.272} C_VEL
LIN {X 0,Y 517.321,Z 1234.018,A -85,B 0,C 180,E1 11788.321,E2 11788.321} C_VEL
LIN {X 0,Y 517.223,Z 1234.015,A -85,B 0,C 180,E1 11791.679,E2 11791.679} C_VEL
LIN {X 0,Y 517.388,Z 1228.998,A -85,B 0,C 180,E1 11796.727,E2 11796.727} C_VEL
LIN {X 0,Y 517.857,Z 1219.129,A -85,B 0,C 180,E1 11801.336,E2 11801.336} C_VEL
LIN {X 0,Y 519.18,Z 1202.909,A -85,B 0,C 180,E1 11806.192,E2 11806.192} C_VEL
LIN {X 0,Y 521.806,Z 1179.492,A -85,B 0,C 180,E1 11811.121,E2 11811.121} C_VEL
LIN {X 0,Y 525.855,Z 1150.76,A -85,B 0,C 180,E1 11815.609,E2 11815.609} C_VEL
LIN {X 0,Y 531.128,Z 1116.353,A -85,B 0,C 180,E1 11819.689,E2 11819.689} C_VEL
LIN {X 0,Y 536.997,Z 1078.22,A -85,B 0,C 180,E1 11823.122,E2 11823.122} C_VEL
LIN {X 0,Y 543.01,Z 1035.465,A -85,B 0,C 180,E1 11825.994,E2 11825.994} C_VEL
LIN {X 0,Y 548.263,Z 990.027,A -85,B 0,C 180,E1 11828.175,E2 11828.175} C_VEL
LIN {X 0,Y 552.292,Z 941.929,A -85,B 0,C 180,E1 11829.676,E2 11829.676} C_VEL
LIN {X 0,Y 551.073,Z 934.419,A -85,B 0,C 180,E1 11829.965,E2 11829.965} C_VEL
LIN {X 0,Y 537.847,Z 902.268,A -85,B 0,C 180,E1 11831.718,E2 11831.718} C_VEL
LIN {X 0,Y 515.943,Z 860.295,A -85,B 0,C 180,E1 11834.497,E2 11834.497} C_VEL
LIN {X 0,Y 515.853,Z 859.31,A -85,B 0,C 180,E1 11834.828,E2 11834.828} C_VEL
LIN {X 0,Y 515.826,Z 859.31,A -85,B 0,C 180,E1 11839.798,E2 11839.798} C_VEL
LIN {X 0,Y 515.844,Z 859.31,A -85,B 0,C 180,E1 11846.081,E2 11846.081} C_VEL
LIN {X 0,Y 516.094,Z 859.31,A -85,B 0,C 180,E1 11851.986,E2 11851.986} C_VEL
LIN {X 0,Y 516.292,Z 859.31,A -85,B 0,C 180,E1 11857.574,E2 11857.574} C_VEL
LIN {X 0,Y 516.443,Z 859.31,A -85,B 0,C 180,E1 11862.94,E2 11862.94} C_VEL
LIN {X 0,Y 516.565,Z 859.31,A -85,B 0,C 180,E1 11868.152,E2 11868.152} C_VEL
LIN {X 0,Y 516.86,Z 859.31,A -85,B 0,C 180,E1 11873.265,E2 11873.265} C_VEL
LIN {X 0,Y 517.038,Z 859.31,A -85,B 0,C 180,E1 11878.319,E2 11878.319} C_VEL
LIN {X 0,Y 517.003,Z 859.31,A -85,B 0,C 180,E1 11883.357,E2 11883.357} C_VEL
LIN {X 0,Y 516.731,Z 859.31,A -85,B 0,C 180,E1 11888.427,E2 11888.427} C_VEL
LIN {X 0,Y 516.506,Z 859.31,A -85,B 0,C 180,E1 11894.504,E2 11894.504} C_VEL
LIN {X 0,Y 516.335,Z 859.31,A -85,B 0,C 180,E1 11900.612,E2 11900.612} C_VEL
LIN {X 0,Y 516.106,Z 859.31,A -85,B 0,C 180,E1 11906.119,E2 11906.119} C_VEL
LIN {X 0,Y 515.971,Z 859.31,A -85,B 0,C 180,E1 11911.9,E2 11911.9} C_VEL
LIN {X 0,Y 515.816,Z 859.31,A -85,B 0,C 180,E1 11918.076,E2 11918.076} C_VEL
LIN {X 0,Y 515.717,Z 859.31,A -85,B 0,C 180,E1 11924.825,E2 11924.825} C_VEL
LIN {X 0,Y 515.82,Z 859.31,A -85,B 0,C 180,E1 11929.778,E2 11929.778} C_VEL
LIN {X 0,Y 515.891,Z 859.353,A -85,B 0,C 180,E1 11931.649,E2 11931.649} C_VEL
LIN {X 0,Y 518.508,Z 865.175,A -85,B 0,C 180,E1 11932.001,E2 11932.001} C_VEL
LIN {X 0,Y 544.757,Z 914.612,A -85,B 0,C 180,E1 11935.116,E2 11935.116} C_VEL
LIN {X 0,Y 552.607,Z 932.327,A -85,B 0,C 180,E1 11936.009,E2 11936.009} C_VEL
LIN {X 0,Y 550.897,Z 975.277,A -85,B 0,C 180,E1 11936.748,E2 11936.748} C_VEL
LIN {X 0,Y 547.403,Z 1012.924,A -85,B 0,C 180,E1 11937.924,E2 11937.924} C_VEL
LIN {X 0,Y 542.571,Z 1049.972,A -85,B 0,C 180,E1 11939.705,E2 11939.705} C_VEL
LIN {X 0,Y 536.935,Z 1085.328,A -85,B 0,C 180,E1 11942.134,E2 11942.134} C_VEL
LIN {X 0,Y 531.218,Z 1117.072,A -85,B 0,C 180,E1 11945.119,E2 11945.119} C_VEL
LIN {X 0,Y 526.212,Z 1143.676,A -85,B 0,C 180,E1 11948.46,E2 11948.46} C_VEL
LIN {X 0,Y 522.016,Z 1167.353,A -85,B 0,C 180,E1 11952.473,E2 11952.473} C_VEL
LIN {X 0,Y 519.267,Z 1185.726,A -85,B 0,C 180,E1 11956.813,E2 11956.813} C_VEL
LIN {X 0,Y 517.996,Z 1197.261,A -85,B 0,C 180,E1 11960.742,E2 11960.742} C_VEL
LIN {X 0,Y 517.476,Z 1204.788,A -85,B 0,C 180,E1 11964.96,E2 11964.96} C_VEL
LIN {X 0,Y 517.279,Z 1207.927,A -85,B 0,C 180,E1 11970,E2 11970} C_VEL
LIN {X 0,Y 517.33,Z 1206.455,A -85,B 0,C 180,E1 11973.359,E2 11973.359} C_VEL
LIN {X 0,Y 517.763,Z 1200.67,A -85,B 0,C 180,E1 11977.568,E2 11977.568} C_VEL
LIN {X 0,Y 518.97,Z 1188.493,A -85,B 0,C 180,E1 11982.288,E2 11982.288} C_VEL
LIN {X 0,Y 521.277,Z 1171.586,A -85,B 0,C 180,E1 11986.574,E2 11986.574} C_VEL
LIN {X 0,Y 525.255,Z 1148.696,A -85,B 0,C 180,E1 11990.695,E2 11990.695} C_VEL
LIN {X 0,Y 530.25,Z 1122.056,A -85,B 0,C 180,E1 11994.232,E2 11994.232} C_VEL
LIN {X 0,Y 535.743,Z 1092.116,A -85,B 0,C 180,E1 11997.209,E2 11997.209} C_VEL
LIN {X 0,Y 541.348,Z 1058.215,A -85,B 0,C 180,E1 11999.705,E2 11999.705} C_VEL
LIN {X 0,Y 546.513,Z 1020.484,A -85,B 0,C 180,E1 12001.673,E2 12001.673} C_VEL
LIN {X 0,Y 550.353,Z 981.054,A -85,B 0,C 180,E1 12003.024,E2 12003.024} C_VEL
LIN {X 0,Y 552.407,Z 937.785,A -85,B 0,C 180,E1 12003.831,E2 12003.831} C_VEL
LIN {X 0,Y 552.006,Z 929.846,A -85,B 0,C 180,E1 12003.977,E2 12003.977} C_VEL
LIN {X 0,Y 527.801,Z 881.948,A -85,B 0,C 180,E1 12006.753,E2 12006.753} C_VEL
LIN {X 0,Y 515.944,Z 860.343,A -85,B 0,C 180,E1 12008.225,E2 12008.225} C_VEL
LIN {X 0,Y 515.866,Z 859.31,A -85,B 0,C 180,E1 12008.456,E2 12008.456} C_VEL
LIN {X 0,Y 515.718,Z 859.31,A -85,B 0,C 180,E1 12014.844,E2 12014.844} C_VEL
LIN {X 0,Y 515.77,Z 859.31,A -85,B 0,C 180,E1 12019.806,E2 12019.806} C_VEL
LIN {X 0,Y 515.884,Z 859.31,A -85,B 0,C 180,E1 12026.09,E2 12026.09} C_VEL
LIN {X 0,Y 516.04,Z 859.31,A -85,B 0,C 180,E1 12031.988,E2 12031.988} C_VEL
LIN {X 0,Y 516.232,Z 859.31,A -85,B 0,C 180,E1 12037.577,E2 12037.577} C_VEL
LIN {X 0,Y 516.236,Z 859.31,A -85,B 0,C 180,E1 12042.938,E2 12042.938} C_VEL
LIN {X 0,Y 516.573,Z 859.31,A -85,B 0,C 180,E1 12048.156,E2 12048.156} C_VEL
LIN {X 0,Y 516.881,Z 859.31,A -85,B 0,C 180,E1 12053.27,E2 12053.27} C_VEL
LIN {X 0,Y 517.041,Z 859.31,A -85,B 0,C 180,E1 12058.323,E2 12058.323} C_VEL
LIN {X 0,Y 517.001,Z 859.31,A -85,B 0,C 180,E1 12063.362,E2 12063.362} C_VEL
LIN {X 0,Y 516.713,Z 859.31,A -85,B 0,C 180,E1 12068.432,E2 12068.432} C_VEL
LIN {X 0,Y 516.472,Z 859.31,A -85,B 0,C 180,E1 12074.488,E2 12074.488} C_VEL
LIN {X 0,Y 516.359,Z 859.31,A -85,B 0,C 180,E1 12080.616,E2 12080.616} C_VEL
LIN {X 0,Y 516.144,Z 859.31,A -85,B 0,C 180,E1 12086.123,E2 12086.123} C_VEL
LIN {X 0,Y 515.984,Z 859.31,A -85,B 0,C 180,E1 12091.905,E2 12091.905} C_VEL
LIN {X 0,Y 515.817,Z 859.31,A -85,B 0,C 180,E1 12098.082,E2 12098.082} C_VEL
LIN {X 0,Y 515.733,Z 859.31,A -85,B 0,C 180,E1 12102.732,E2 12102.732} C_VEL
LIN {X 0,Y 515.755,Z 860.009,A -85,B 0,C 180,E1 12105.491,E2 12105.491} C_VEL
LIN {X 0,Y 542.206,Z 911.538,A -85,B 0,C 180,E1 12108.821,E2 12108.821} C_VEL
LIN {X 0,Y 552.519,Z 939.679,A -85,B 0,C 180,E1 12110.289,E2 12110.289} C_VEL
LIN {X 0,Y 548.941,Z 981.917,A -85,B 0,C 180,E1 12111.525,E2 12111.525} C_VEL
LIN {X 0,Y 544.493,Z 1023.699,A -85,B 0,C 180,E1 12113.374,E2 12113.374} C_VEL
LIN {X 0,Y 538.809,Z 1065.615,A -85,B 0,C 180,E1 12115.942,E2 12115.942} C_VEL
LIN {X 0,Y 532.84,Z 1105.195,A -85,B 0,C 180,E1 12119.21,E2 12119.21} C_VEL
LIN {X 0,Y 527.437,Z 1140.259,A -85,B 0,C 180,E1 12123.027,E2 12123.027} C_VEL
LIN {X 0,Y 522.908,Z 1171.03,A -85,B 0,C 180,E1 12127.42,E2 12127.42} C_VEL
LIN {X 0,Y 521.771,Z 1179.869,A -85,B 0,C 180,E1 12128.95,E2 12128.95} C_VEL
LIN {X 0,Y 519.992,Z 1184.358,A -85,B 0,C 180,E1 12129.756,E2 12129.756} C_VEL
LIN {X 0,Y 512.055,Z 1195.918,A -85,B 0,C 180,E1 12131.958,E2 12131.958} C_VEL
LIN {X 0,Y 511.891,Z 1196.844,A -85,B 0,C 180,E1 12132.178,E2 12132.178} C_VEL
LIN {X 0,Y 510.244,Z 1215.033,A -85,B 0,C 180,E1 12137.13,E2 12137.13} C_VEL
LIN {X 0,Y 509.596,Z 1225.71,A -85,B 0,C 180,E1 12141.45,E2 12141.45} C_VEL
LIN {X 0,Y 509.437,Z 1231.11,A -85,B 0,C 180,E1 12144.88,E2 12144.88} C_VEL
LIN {X 0,Y 509.417,Z 1233.814,A -85,B 0,C 180,E1 12148.295,E2 12148.295} C_VEL
LIN {X 0,Y 509.324,Z 1233.812,A -85,B 0,C 180,E1 12151.705,E2 12151.705} C_VEL
LIN {X 0,Y 509.466,Z 1230.025,A -85,B 0,C 180,E1 12155.975,E2 12155.975} C_VEL
LIN {X 0,Y 509.922,Z 1220.64,A -85,B 0,C 180,E1 12160.835,E2 12160.835} C_VEL
LIN {X 0,Y 511.039,Z 1206.199,A -85,B 0,C 180,E1 12165.477,E2 12165.477} C_VEL
LIN {X 0,Y 513.218,Z 1186.278,A -85,B 0,C 180,E1 12170.074,E2 12170.074} C_VEL
LIN {X 0,Y 516.884,Z 1160.147,A -85,B 0,C 180,E1 12174.588,E2 12174.588} C_VEL
LIN {X 0,Y 522.023,Z 1127.583,A -85,B 0,C 180,E1 12178.854,E2 12178.854} C_VEL
LIN {X 0,Y 528.035,Z 1090.888,A -85,B 0,C 180,E1 12182.509,E2 12182.509} C_VEL
LIN {X 0,Y 534.308,Z 1049.336,A -85,B 0,C 180,E1 12185.62,E2 12185.62} C_VEL
LIN {X 0,Y 540.154,Z 1004.498,A -85,B 0,C 180,E1 12188.045,E2 12188.045} C_VEL
LIN {X 0,Y 544.78,Z 958.3,A -85,B 0,C 180,E1 12189.737,E2 12189.737} C_VEL
LIN {X 0,Y 545.505,Z 939.379,A -85,B 0,C 180,E1 12190.272,E2 12190.272} C_VEL
LIN {X 0,Y 533.539,Z 909.05,A -85,B 0,C 180,E1 12191.962,E2 12191.962} C_VEL
LIN {X 0,Y 512.44,Z 869.045,A -85,B 0,C 180,E1 12194.668,E2 12194.668} C_VEL
LIN {X 0,Y 508.01,Z 860.236,A -85,B 0,C 180,E1 12195.289,E2 12195.289} C_VEL
LIN {X 0,Y 507.915,Z 859.31,A -85,B 0,C 180,E1 12195.419,E2 12195.419} C_VEL
LIN {X 0,Y 507.843,Z 859.31,A -85,B 0,C 180,E1 12201.21,E2 12201.21} C_VEL
LIN {X 0,Y 507.973,Z 859.31,A -85,B 0,C 180,E1 12207.531,E2 12207.531} C_VEL
LIN {X 0,Y 508.225,Z 859.31,A -85,B 0,C 180,E1 12213.439,E2 12213.439} C_VEL
LIN {X 0,Y 508.406,Z 859.31,A -85,B 0,C 180,E1 12219.047,E2 12219.047} C_VEL
LIN {X 0,Y 508.528,Z 859.31,A -85,B 0,C 180,E1 12224.446,E2 12224.446} C_VEL
LIN {X 0,Y 508.731,Z 859.31,A -85,B 0,C 180,E1 12229.706,E2 12229.706} C_VEL
LIN {X 0,Y 509.029,Z 859.31,A -85,B 0,C 180,E1 12234.875,E2 12234.875} C_VEL
LIN {X 0,Y 509.253,Z 859.31,A -85,B 0,C 180,E1 12239.998,E2 12239.998} C_VEL
LIN {X 0,Y 509.076,Z 859.31,A -85,B 0,C 180,E1 12245.119,E2 12245.119} C_VEL
LIN {X 0,Y 508.726,Z 859.31,A -85,B 0,C 180,E1 12250.6,E2 12250.6} C_VEL
LIN {X 0,Y 508.555,Z 859.31,A -85,B 0,C 180,E1 12255.548,E2 12255.548} C_VEL
LIN {X 0,Y 508.38,Z 859.31,A -85,B 0,C 180,E1 12260.949,E2 12260.949} C_VEL
LIN {X 0,Y 508.167,Z 859.31,A -85,B 0,C 180,E1 12266.559,E2 12266.559} C_VEL
LIN {X 0,Y 507.978,Z 859.31,A -85,B 0,C 180,E1 12272.463,E2 12272.463} C_VEL
LIN {X 0,Y 507.821,Z 859.31,A -85,B 0,C 180,E1 12278.786,E2 12278.786} C_VEL
LIN {X 0,Y 507.774,Z 859.31,A -85,B 0,C 180,E1 12284.258,E2 12284.258} C_VEL
LIN {X 0,Y 507.904,Z 859.408,A -85,B 0,C 180,E1 12290.845,E2 12290.845} C_VEL
LIN {X 0,Y 510.354,Z 864.979,A -85,B 0,C 180,E1 12291.19,E2 12291.19} C_VEL
LIN {X 0,Y 535.03,Z 910.271,A -85,B 0,C 180,E1 12294.227,E2 12294.227} C_VEL
LIN {X 0,Y 546.203,Z 933.617,A -85,B 0,C 180,E1 12295.514,E2 12295.514} C_VEL
LIN {X 0,Y 544.432,Z 976.573,A -85,B 0,C 180,E1 12296.285,E2 12296.285} C_VEL
LIN {X 0,Y 540.835,Z 1013.504,A -85,B 0,C 180,E1 12297.464,E2 12297.464} C_VEL
LIN {X 0,Y 535.809,Z 1050.667,A -85,B 0,C 180,E1 12299.282,E2 12299.282} C_VEL
LIN {X 0,Y 529.962,Z 1085.841,A -85,B 0,C 180,E1 12301.734,E2 12301.734} C_VEL
LIN {X 0,Y 524.016,Z 1117.476,A -85,B 0,C 180,E1 12304.753,E2 12304.753} C_VEL
LIN {X 0,Y 518.805,Z 1144.009,A -85,B 0,C 180,E1 12308.137,E2 12308.137} C_VEL
LIN {X 0,Y 514.394,Z 1167.638,A -85,B 0,C 180,E1 12312.204,E2 12312.204} C_VEL
LIN {X 0,Y 511.622,Z 1184.91,A -85,B 0,C 180,E1 12316.294,E2 12316.294} C_VEL
LIN {X 0,Y 510.163,Z 1197.486,A -85,B 0,C 180,E1 12320.598,E2 12320.598} C_VEL
LIN {X 0,Y 509.591,Z 1204.998,A -85,B 0,C 180,E1 12324.882,E2 12324.882} C_VEL
LIN {X 0,Y 509.364,Z 1207.798,A -85,B 0,C 180,E1 12328.295,E2 12328.295} C_VEL
LIN {X 0,Y 509.45,Z 1207.742,A -85,B 0,C 180,E1 12331.705,E2 12331.705} C_VEL
LIN {X 0,Y 509.621,Z 1204.116,A -85,B 0,C 180,E1 12335.686,E2 12335.686} C_VEL
LIN {X 0,Y 510.372,Z 1195.088,A -85,B 0,C 180,E1 12340.262,E2 12340.262} C_VEL
LIN {X 0,Y 512.166,Z 1181.348,A -85,B 0,C 180,E1 12344.565,E2 12344.565} C_VEL
LIN {X 0,Y 515.215,Z 1162.752,A -85,B 0,C 180,E1 12348.654,E2 12348.654} C_VEL
LIN {X 0,Y 519.74,Z 1139.004,A -85,B 0,C 180,E1 12352.481,E2 12352.481} C_VEL
LIN {X 0,Y 525.238,Z 1110.979,A -85,B 0,C 180,E1 12355.849,E2 12355.849} C_VEL
LIN {X 0,Y 531.054,Z 1079.578,A -85,B 0,C 180,E1 12358.668,E2 12358.668} C_VEL
LIN {X 0,Y 536.606,Z 1045.733,A -85,B 0,C 180,E1 12360.903,E2 12360.903} C_VEL
LIN {X 0,Y 541.479,Z 1007.959,A -85,B 0,C 180,E1 12362.657,E2 12362.657} C_VEL
LIN {X 0,Y 544.985,Z 967.106,A -85,B 0,C 180,E1 12363.846,E2 12363.846} C_VEL
LIN {X 0,Y 545.568,Z 932.109,A -85,B 0,C 180,E1 12364.461,E2 12364.461} C_VEL
LIN {X 0,Y 521.698,Z 884.959,A -85,B 0,C 180,E1 12367.272,E2 12367.272} C_VEL
LIN {X 0,Y 508.015,Z 860.596,A -85,B 0,C 180,E1 12369.017,E2 12369.017} C_VEL
LIN {X 0,Y 507.893,Z 859.31,A -85,B 0,C 180,E1 12369.153,E2 12369.153} C_VEL
LIN {X 0,Y 507.775,Z 859.31,A -85,B 0,C 180,E1 12375.742,E2 12375.742} C_VEL
LIN {X 0,Y 507.831,Z 859.31,A -85,B 0,C 180,E1 12381.215,E2 12381.215} C_VEL
LIN {X 0,Y 507.973,Z 859.31,A -85,B 0,C 180,E1 12386.642,E2 12386.642} C_VEL
LIN {X 0,Y 508.123,Z 859.31,A -85,B 0,C 180,E1 12391.512,E2 12391.512} C_VEL
LIN {X 0,Y 508.329,Z 859.31,A -85,B 0,C 180,E1 12397.532,E2 12397.532} C_VEL
LIN {X 0,Y 508.297,Z 859.31,A -85,B 0,C 180,E1 12402.663,E2 12402.663} C_VEL
LIN {X 0,Y 508.649,Z 859.31,A -85,B 0,C 180,E1 12407.969,E2 12407.969} C_VEL
LIN {X 0,Y 508.962,Z 859.31,A -85,B 0,C 180,E1 12413.165,E2 12413.165} C_VEL
LIN {X 0,Y 509.152,Z 859.31,A -85,B 0,C 180,E1 12418.297,E2 12418.297} C_VEL
LIN {X 0,Y 509.113,Z 859.31,A -85,B 0,C 180,E1 12423.414,E2 12423.414} C_VEL
LIN {X 0,Y 508.793,Z 859.31,A -85,B 0,C 180,E1 12428.564,E2 12428.564} C_VEL
LIN {X 0,Y 508.593,Z 859.31,A -85,B 0,C 180,E1 12433.788,E2 12433.788} C_VEL
LIN {X 0,Y 508.476,Z 859.31,A -85,B 0,C 180,E1 12439.133,E2 12439.133} C_VEL
LIN {X 0,Y 508.246,Z 859.31,A -85,B 0,C 180,E1 12444.666,E2 12444.666} C_VEL
LIN {X 0,Y 508.104,Z 859.31,A -85,B 0,C 180,E1 12450.457,E2 12450.457} C_VEL
LIN {X 0,Y 507.912,Z 859.31,A -85,B 0,C 180,E1 12456.624,E2 12456.624} C_VEL
LIN {X 0,Y 507.768,Z 859.31,A -85,B 0,C 180,E1 12463.332,E2 12463.332} C_VEL
LIN {X 0,Y 507.791,Z 859.31,A -85,B 0,C 180,E1 12464.667,E2 12464.667} C_VEL
LIN {X 0,Y 510.315,Z 865.086,A -85,B 0,C 180,E1 12465.053,E2 12465.053} C_VEL
LIN {X 0,Y 534.436,Z 910.99,A -85,B 0,C 180,E1 12468.159,E2 12468.159} C_VEL
LIN {X 0,Y 545.968,Z 940.848,A -85,B 0,C 180,E1 12469.81,E2 12469.81} C_VEL
LIN {X 0,Y 542.161,Z 985.545,A -85,B 0,C 180,E1 12471.177,E2 12471.177} C_VEL
LIN {X 0,Y 537.455,Z 1026.692,A -85,B 0,C 180,E1 12473.067,E2 12473.067} C_VEL
LIN {X 0,Y 531.651,Z 1067.334,A -85,B 0,C 180,E1 12475.624,E2 12475.624} C_VEL
LIN {X 0,Y 525.632,Z 1105.718,A -85,B 0,C 180,E1 12478.857,E2 12478.857} C_VEL
LIN {X 0,Y 520.114,Z 1139.807,A -85,B 0,C 180,E1 12482.615,E2 12482.615} C_VEL
LIN {X 0,Y 515.342,Z 1170.638,A -85,B 0,C 180,E1 12487.07,E2 12487.07} C_VEL
LIN {X 0,Y 512.195,Z 1193.755,A -85,B 0,C 180,E1 12491.489,E2 12491.489} C_VEL
LIN {X 0,Y 511.891,Z 1196.844,A -85,B 0,C 180,E1 12492.178,E2 12492.178} C_VEL
LIN {X 0,Y 508.946,Z 1202.467,A -85,B 0,C 180,E1 12493.473,E2 12493.473} C_VEL
LIN {X 0,Y 502.873,Z 1210.021,A -85,B 0,C 180,E1 12495.439,E2 12495.439} C_VEL
LIN {X 0,Y 502.694,Z 1210.769,A -85,B 0,C 180,E1 12495.674,E2 12495.674} C_VEL
LIN {X 0,Y 501.822,Z 1223.722,A -85,B 0,C 180,E1 12500.44,E2 12500.44} C_VEL
LIN {X 0,Y 501.551,Z 1230.892,A -85,B 0,C 180,E1 12504.8,E2 12504.8} C_VEL
LIN {X 0,Y 501.514,Z 1233.61,A -85,B 0,C 180,E1 12508.268,E2 12508.268} C_VEL
LIN {X 0,Y 501.424,Z 1233.608,A -85,B 0,C 180,E1 12511.732,E2 12511.732} C_VEL
LIN {X 0,Y 501.58,Z 1229.798,A -85,B 0,C 180,E1 12516.069,E2 12516.069} C_VEL
LIN {X 0,Y 502.06,Z 1220.382,A -85,B 0,C 180,E1 12521.007,E2 12521.007} C_VEL
LIN {X 0,Y 503.235,Z 1205.899,A -85,B 0,C 180,E1 12525.724,E2 12525.724} C_VEL
LIN {X 0,Y 505.612,Z 1185.934,A -85,B 0,C 180,E1 12530.389,E2 12530.389} C_VEL
LIN {X 0,Y 509.326,Z 1160.466,A -85,B 0,C 180,E1 12534.866,E2 12534.866} C_VEL
LIN {X 0,Y 514.51,Z 1129.029,A -85,B 0,C 180,E1 12539.074,E2 12539.074} C_VEL
LIN {X 0,Y 520.763,Z 1092.478,A -85,B 0,C 180,E1 12542.801,E2 12542.801} C_VEL
LIN {X 0,Y 527.271,Z 1051.355,A -85,B 0,C 180,E1 12545.957,E2 12545.957} C_VEL
LIN {X 0,Y 533.348,Z 1006.958,A -85,B 0,C 180,E1 12548.425,E2 12548.425} C_VEL
LIN {X 0,Y 538.195,Z 961.099,A -85,B 0,C 180,E1 12550.155,E2 12550.155} C_VEL
LIN {X 0,Y 539.152,Z 941.948,A -85,B 0,C 180,E1 12550.715,E2 12550.715} C_VEL
LIN {X 0,Y 527.668,Z 912.675,A -85,B 0,C 180,E1 12552.405,E2 12552.405} C_VEL
LIN {X 0,Y 505.561,Z 870.41,A -85,B 0,C 180,E1 12555.334,E2 12555.334} C_VEL
LIN {X 0,Y 500.069,Z 860.406,A -85,B 0,C 180,E1 12556.114,E2 12556.114} C_VEL
LIN {X 0,Y 499.993,Z 859.31,A -85,B 0,C 180,E1 12556.275,E2 12556.275} C_VEL
LIN {X 0,Y 499.898,Z 859.31,A -85,B 0,C 180,E1 12562.691,E2 12562.691} C_VEL
LIN {X 0,Y 500.107,Z 859.31,A -85,B 0,C 180,E1 12569.003,E2 12569.003} C_VEL
LIN {X 0,Y 500.391,Z 859.31,A -85,B 0,C 180,E1 12575.294,E2 12575.294} C_VEL
LIN {X 0,Y 500.519,Z 859.31,A -85,B 0,C 180,E1 12580.551,E2 12580.551} C_VEL
LIN {X 0,Y 500.624,Z 859.31,A -85,B 0,C 180,E1 12585.988,E2 12585.988} C_VEL
LIN {X 0,Y 500.914,Z 859.31,A -85,B 0,C 180,E1 12591.3,E2 12591.3} C_VEL
LIN {X 0,Y 501.22,Z 859.31,A -85,B 0,C 180,E1 12596.532,E2 12596.532} C_VEL
LIN {X 0,Y 501.336,Z 859.31,A -85,B 0,C 180,E1 12601.729,E2 12601.729} C_VEL
LIN {X 0,Y 501.023,Z 859.31,A -85,B 0,C 180,E1 12606.944,E2 12606.944} C_VEL
LIN {X 0,Y 500.755,Z 859.31,A -85,B 0,C 180,E1 12612.223,E2 12612.223} C_VEL
LIN {X 0,Y 500.588,Z 859.31,A -85,B 0,C 180,E1 12617.613,E2 12617.613} C_VEL
LIN {X 0,Y 500.328,Z 859.31,A -85,B 0,C 180,E1 12623.177,E2 12623.177} C_VEL
LIN {X 0,Y 500.183,Z 859.31,A -85,B 0,C 180,E1 12628.983,E2 12628.983} C_VEL
LIN {X 0,Y 500.009,Z 859.31,A -85,B 0,C 180,E1 12635.142,E2 12635.142} C_VEL
LIN {X 0,Y 499.889,Z 859.31,A -85,B 0,C 180,E1 12641.81,E2 12641.81} C_VEL
LIN {X 0,Y 499.909,Z 859.31,A -85,B 0,C 180,E1 12648.176,E2 12648.176} C_VEL
LIN {X 0,Y 500.025,Z 859.31,A -85,B 0,C 180,E1 12650.004,E2 12650.004} C_VEL
LIN {X 0,Y 502.41,Z 864.998,A -85,B 0,C 180,E1 12650.368,E2 12650.368} C_VEL
LIN {X 0,Y 527.679,Z 910.53,A -85,B 0,C 180,E1 12653.581,E2 12653.581} C_VEL
LIN {X 0,Y 540,Z 937.772,A -85,B 0,C 180,E1 12655.064,E2 12655.064} C_VEL
LIN {X 0,Y 537.764,Z 981.132,A -85,B 0,C 180,E1 12655.893,E2 12655.893} C_VEL
LIN {X 0,Y 533.581,Z 1020.232,A -85,B 0,C 180,E1 12657.251,E2 12657.251} C_VEL
LIN {X 0,Y 528.019,Z 1058.258,A -85,B 0,C 180,E1 12659.271,E2 12659.271} C_VEL
LIN {X 0,Y 521.632,Z 1093.738,A -85,B 0,C 180,E1 12661.951,E2 12661.951} C_VEL
LIN {X 0,Y 515.326,Z 1125.229,A -85,B 0,C 180,E1 12665.228,E2 12665.228} C_VEL
LIN {X 0,Y 509.738,Z 1152.582,A -85,B 0,C 180,E1 12669.101,E2 12669.101} C_VEL
LIN {X 0,Y 505.779,Z 1173.647,A -85,B 0,C 180,E1 12673.16,E2 12673.16} C_VEL
LIN {X 0,Y 503.3,Z 1189.504,A -85,B 0,C 180,E1 12677.392,E2 12677.392} C_VEL
LIN {X 0,Y 501.949,Z 1201.264,A -85,B 0,C 180,E1 12682.193,E2 12682.193} C_VEL
LIN {X 0,Y 501.559,Z 1206.956,A -85,B 0,C 180,E1 12686.536,E2 12686.536} C_VEL
LIN {X 0,Y 501.484,Z 1208.331,A -85,B 0,C 180,E1 12690,E2 12690} C_VEL
LIN {X 0,Y 501.679,Z 1205.558,A -85,B 0,C 180,E1 12694.837,E2 12694.837} C_VEL
LIN {X 0,Y 502.358,Z 1197.492,A -85,B 0,C 180,E1 12699.55,E2 12699.55} C_VEL
LIN {X 0,Y 504.203,Z 1183.263,A -85,B 0,C 180,E1 12704.356,E2 12704.356} C_VEL
LIN {X 0,Y 507.425,Z 1164.205,A -85,B 0,C 180,E1 12708.725,E2 12708.725} C_VEL
LIN {X 0,Y 512.091,Z 1140.787,A -85,B 0,C 180,E1 12712.624,E2 12712.624} C_VEL
LIN {X 0,Y 517.739,Z 1113.262,A -85,B 0,C 180,E1 12716.041,E2 12716.041} C_VEL
LIN {X 0,Y 524.147,Z 1080.142,A -85,B 0,C 180,E1 12719.081,E2 12719.081} C_VEL
LIN {X 0,Y 530.142,Z 1044.643,A -85,B 0,C 180,E1 12721.442,E2 12721.442} C_VEL
LIN {X 0,Y 535.15,Z 1006.651,A -85,B 0,C 180,E1 12723.201,E2 12723.201} C_VEL
LIN {X 0,Y 538.778,Z 965.919,A -85,B 0,C 180,E1 12724.374,E2 12724.374} C_VEL
LIN {X 0,Y 539.293,Z 934.791,A -85,B 0,C 180,E1 12724.94,E2 12724.94} C_VEL
LIN {X 0,Y 516.454,Z 889.461,A -85,B 0,C 180,E1 12727.698,E2 12727.698} C_VEL
LIN {X 0,Y 500.039,Z 860.793,A -85,B 0,C 180,E1 12729.851,E2 12729.851} C_VEL
LIN {X 0,Y 499.891,Z 859.31,A -85,B 0,C 180,E1 12729.977,E2 12729.977} C_VEL
LIN {X 0,Y 499.871,Z 859.31,A -85,B 0,C 180,E1 12735.814,E2 12735.814} C_VEL
LIN {X 0,Y 499.907,Z 859.31,A -85,B 0,C 180,E1 12742.009,E2 12742.009} C_VEL
LIN {X 0,Y 500.053,Z 859.31,A -85,B 0,C 180,E1 12748.046,E2 12748.046} C_VEL
LIN {X 0,Y 500.208,Z 859.31,A -85,B 0,C 180,E1 12752.984,E2 12752.984} C_VEL
LIN {X 0,Y 500.372,Z 859.31,A -85,B 0,C 180,E1 12758.699,E2 12758.699} C_VEL
LIN {X 0,Y 500.443,Z 859.31,A -85,B 0,C 180,E1 12764.193,E2 12764.193} C_VEL
LIN {X 0,Y 500.854,Z 859.31,A -85,B 0,C 180,E1 12769.547,E2 12769.547} C_VEL
LIN {X 0,Y 501.144,Z 859.31,A -85,B 0,C 180,E1 12774.799,E2 12774.799} C_VEL
LIN {X 0,Y 501.359,Z 859.31,A -85,B 0,C 180,E1 12780.002,E2 12780.002} C_VEL
LIN {X 0,Y 501.169,Z 859.31,A -85,B 0,C 180,E1 12785.205,E2 12785.205} C_VEL
LIN {X 0,Y 500.845,Z 859.31,A -85,B 0,C 180,E1 12790.458,E2 12790.458} C_VEL
LIN {X 0,Y 500.642,Z 859.31,A -85,B 0,C 180,E1 12795.805,E2 12795.805} C_VEL
LIN {X 0,Y 500.503,Z 859.31,A -85,B 0,C 180,E1 12801.3,E2 12801.3} C_VEL
LIN {X 0,Y 500.23,Z 859.31,A -85,B 0,C 180,E1 12807.02,E2 12807.02} C_VEL
LIN {X 0,Y 500.063,Z 859.31,A -85,B 0,C 180,E1 12813.047,E2 12813.047} C_VEL
LIN {X 0,Y 499.88,Z 859.31,A -85,B 0,C 180,E1 12819.527,E2 12819.527} C_VEL
LIN {X 0,Y 499.881,Z 859.31,A -85,B 0,C 180,E1 12823.84,E2 12823.84} C_VEL
LIN {X 0,Y 502.491,Z 865.191,A -85,B 0,C 180,E1 12824.254,E2 12824.254} C_VEL
LIN {X 0,Y 526.405,Z 910.043,A -85,B 0,C 180,E1 12827.441,E2 12827.441} C_VEL
LIN {X 0,Y 538.441,Z 939.807,A -85,B 0,C 180,E1 12829.177,E2 12829.177} C_VEL
LIN {X 0,Y 539.52,Z 944.916,A -85,B 0,C 180,E1 12829.413,E2 12829.413} C_VEL
LIN {X 0,Y 535.408,Z 988.934,A -85,B 0,C 180,E1 12830.809,E2 12830.809} C_VEL
LIN {X 0,Y 530.175,Z 1031.662,A -85,B 0,C 180,E1 12832.859,E2 12832.859} C_VEL
LIN {X 0,Y 524.197,Z 1071.041,A -85,B 0,C 180,E1 12835.448,E2 12835.448} C_VEL
LIN {X 0,Y 518.223,Z 1107.422,A -85,B 0,C 180,E1 12838.611,E2 12838.611} C_VEL
LIN {X 0,Y 512.425,Z 1141.63,A -85,B 0,C 180,E1 12842.491,E2 12842.491} C_VEL
LIN {X 0,Y 507.617,Z 1171.54,A -85,B 0,C 180,E1 12846.933,E2 12846.933} C_VEL
LIN {X 0,Y 504.218,Z 1195.706,A -85,B 0,C 180,E1 12851.695,E2 12851.695} C_VEL
LIN {X 0,Y 502.694,Z 1210.769,A -85,B 0,C 180,E1 12855.674,E2 12855.674} C_VEL
LIN {X 0,Y 498.291,Z 1216.513,A -85,B 0,C 180,E1 12857.504,E2 12857.504} C_VEL
LIN {X 0,Y 494.083,Z 1221.444,A -85,B 0,C 180,E1 12859.392,E2 12859.392} C_VEL
LIN {X 0,Y 493.69,Z 1229.575,A -85,B 0,C 180,E1 12863.833,E2 12863.833} C_VEL
LIN {X 0,Y 493.634,Z 1233.408,A -85,B 0,C 180,E1 12868.241,E2 12868.241} C_VEL
LIN {X 0,Y 493.551,Z 1233.406,A -85,B 0,C 180,E1 12871.759,E2 12871.759} C_VEL
LIN {X 0,Y 493.688,Z 1229.578,A -85,B 0,C 180,E1 12876.167,E2 12876.167} C_VEL
LIN {X 0,Y 494.187,Z 1220.113,A -85,B 0,C 180,E1 12881.194,E2 12881.194} C_VEL
LIN {X 0,Y 495.434,Z 1205.613,A -85,B 0,C 180,E1 12885.978,E2 12885.978} C_VEL
LIN {X 0,Y 497.985,Z 1185.604,A -85,B 0,C 180,E1 12890.715,E2 12890.715} C_VEL
LIN {X 0,Y 502.019,Z 1159.251,A -85,B 0,C 180,E1 12895.384,E2 12895.384} C_VEL
LIN {X 0,Y 507.547,Z 1127.682,A -85,B 0,C 180,E1 12899.63,E2 12899.63} C_VEL
LIN {X 0,Y 514.069,Z 1091.102,A -85,B 0,C 180,E1 12903.373,E2 12903.373} C_VEL
LIN {X 0,Y 520.881,Z 1049.487,A -85,B 0,C 180,E1 12906.561,E2 12906.561} C_VEL
LIN {X 0,Y 527.163,Z 1005.001,A -85,B 0,C 180,E1 12909.016,E2 12909.016} C_VEL
LIN {X 0,Y 532.149,Z 958.511,A -85,B 0,C 180,E1 12910.748,E2 12910.748} C_VEL
LIN {X 0,Y 532.518,Z 943.671,A -85,B 0,C 180,E1 12911.216,E2 12911.216} C_VEL
LIN {X 0,Y 520.975,Z 914.361,A -85,B 0,C 180,E1 12912.971,E2 12912.971} C_VEL
LIN {X 0,Y 500.015,Z 874.728,A -85,B 0,C 180,E1 12915.824,E2 12915.824} C_VEL
LIN {X 0,Y 492.128,Z 860.411,A -85,B 0,C 180,E1 12916.981,E2 12916.981} C_VEL
LIN {X 0,Y 492.048,Z 859.31,A -85,B 0,C 180,E1 12917.167,E2 12917.167} C_VEL
LIN {X 0,Y 491.96,Z 859.31,A -85,B 0,C 180,E1 12923.209,E2 12923.209} C_VEL
LIN {X 0,Y 492.179,Z 859.31,A -85,B 0,C 180,E1 12929.547,E2 12929.547} C_VEL
LIN {X 0,Y 492.358,Z 859.31,A -85,B 0,C 180,E1 12934.482,E2 12934.482} C_VEL
LIN {X 0,Y 492.599,Z 859.31,A -85,B 0,C 180,E1 12940.225,E2 12940.225} C_VEL
LIN {X 0,Y 492.714,Z 859.31,A -85,B 0,C 180,E1 12945.759,E2 12945.759} C_VEL
LIN {X 0,Y 492.989,Z 859.31,A -85,B 0,C 180,E1 12951.159,E2 12951.159} C_VEL
LIN {X 0,Y 493.335,Z 859.31,A -85,B 0,C 180,E1 12956.477,E2 12956.477} C_VEL
LIN {X 0,Y 493.442,Z 859.31,A -85,B 0,C 180,E1 12961.757,E2 12961.757} C_VEL
LIN {X 0,Y 493.1,Z 859.31,A -85,B 0,C 180,E1 12967.056,E2 12967.056} C_VEL
LIN {X 0,Y 492.823,Z 859.31,A -85,B 0,C 180,E1 12972.423,E2 12972.423} C_VEL
LIN {X 0,Y 492.647,Z 859.31,A -85,B 0,C 180,E1 12977.906,E2 12977.906} C_VEL
LIN {X 0,Y 492.404,Z 859.31,A -85,B 0,C 180,E1 12983.572,E2 12983.572} C_VEL
LIN {X 0,Y 492.201,Z 859.31,A -85,B 0,C 180,E1 12989.499,E2 12989.499} C_VEL
LIN {X 0,Y 492.003,Z 859.31,A -85,B 0,C 180,E1 12995.801,E2 12995.801} C_VEL
LIN {X 0,Y 491.956,Z 859.31,A -85,B 0,C 180,E1 13002.334,E2 13002.334} C_VEL
LIN {X 0,Y 492.032,Z 859.31,A -85,B 0,C 180,E1 13009.09,E2 13009.09} C_VEL
LIN {X 0,Y 494.713,Z 865.212,A -85,B 0,C 180,E1 13009.539,E2 13009.539} C_VEL
LIN {X 0,Y 519.411,Z 909.288,A -85,B 0,C 180,E1 13012.801,E2 13012.801} C_VEL
LIN {X 0,Y 533.793,Z 939.348,A -85,B 0,C 180,E1 13014.562,E2 13014.562} C_VEL
LIN {X 0,Y 531.356,Z 982.743,A -85,B 0,C 180,E1 13015.421,E2 13015.421} C_VEL
LIN {X 0,Y 526.785,Z 1023.008,A -85,B 0,C 180,E1 13016.871,E2 13016.871} C_VEL
LIN {X 0,Y 520.824,Z 1061.323,A -85,B 0,C 180,E1 13018.989,E2 13018.989} C_VEL
LIN {X 0,Y 514.4,Z 1095.324,A -85,B 0,C 180,E1 13021.641,E2 13021.641} C_VEL
LIN {X 0,Y 508.091,Z 1125.591,A -85,B 0,C 180,E1 13024.851,E2 13024.851} C_VEL
LIN {X 0,Y 502.542,Z 1151.608,A -85,B 0,C 180,E1 13028.556,E2 13028.556} C_VEL
LIN {X 0,Y 498.209,Z 1173.505,A -85,B 0,C 180,E1 13032.798,E2 13032.798} C_VEL
LIN {X 0,Y 495.506,Z 1189.737,A -85,B 0,C 180,E1 13037.191,E2 13037.191} C_VEL
LIN {X 0,Y 494.084,Z 1201.478,A -85,B 0,C 180,E1 13042.068,E2 13042.068} C_VEL
LIN {X 0,Y 493.662,Z 1207.161,A -85,B 0,C 180,E1 13046.481,E2 13046.481} C_VEL
LIN {X 0,Y 493.6,Z 1208.533,A -85,B 0,C 180,E1 13050,E2 13050} C_VEL
LIN {X 0,Y 493.66,Z 1207.073,A -85,B 0,C 180,E1 13053.52,E2 13053.52} C_VEL
LIN {X 0,Y 494.151,Z 1201.318,A -85,B 0,C 180,E1 13057.932,E2 13057.932} C_VEL
LIN {X 0,Y 495.583,Z 1189.456,A -85,B 0,C 180,E1 13062.808,E2 13062.808} C_VEL
LIN {X 0,Y 498.415,Z 1171.993,A -85,B 0,C 180,E1 13067.455,E2 13067.455} C_VEL
LIN {X 0,Y 502.946,Z 1149.694,A -85,B 0,C 180,E1 13071.659,E2 13071.659} C_VEL
LIN {X 0,Y 508.621,Z 1123.079,A -85,B 0,C 180,E1 13075.358,E2 13075.358} C_VEL
LIN {X 0,Y 515.049,Z 1091.999,A -85,B 0,C 180,E1 13078.56,E2 13078.56} C_VEL
LIN {X 0,Y 521.269,Z 1058.333,A -85,B 0,C 180,E1 13081.116,E2 13081.116} C_VEL
LIN {X 0,Y 527.126,Z 1019.524,A -85,B 0,C 180,E1 13083.19,E2 13083.19} C_VEL
LIN {X 0,Y 531.471,Z 979.963,A -85,B 0,C 180,E1 13084.559,E2 13084.559} C_VEL
LIN {X 0,Y 533.445,Z 938.23,A -85,B 0,C 180,E1 13085.384,E2 13085.384} C_VEL
LIN {X 0,Y 511.395,Z 894.313,A -85,B 0,C 180,E1 13088.111,E2 13088.111} C_VEL
LIN {X 0,Y 492.207,Z 861.037,A -85,B 0,C 180,E1 13090.707,E2 13090.707} C_VEL
LIN {X 0,Y 492.036,Z 859.31,A -85,B 0,C 180,E1 13090.789,E2 13090.789} C_VEL
LIN {X 0,Y 491.952,Z 859.31,A -85,B 0,C 180,E1 13097.358,E2 13097.358} C_VEL
LIN {X 0,Y 492,Z 859.31,A -85,B 0,C 180,E1 13103.204,E2 13103.204} C_VEL
LIN {X 0,Y 492.159,Z 859.31,A -85,B 0,C 180,E1 13109.552,E2 13109.552} C_VEL
LIN {X 0,Y 492.317,Z 859.31,A -85,B 0,C 180,E1 13114.485,E2 13114.485} C_VEL
LIN {X 0,Y 492.43,Z 859.31,A -85,B 0,C 180,E1 13120.223,E2 13120.223} C_VEL
LIN {X 0,Y 492.617,Z 859.31,A -85,B 0,C 180,E1 13125.761,E2 13125.761} C_VEL
LIN {X 0,Y 493.054,Z 859.31,A -85,B 0,C 180,E1 13131.165,E2 13131.165} C_VEL
LIN {X 0,Y 493.34,Z 859.31,A -85,B 0,C 180,E1 13136.481,E2 13136.481} C_VEL
LIN {X 0,Y 493.446,Z 859.31,A -85,B 0,C 180,E1 13141.762,E2 13141.762} C_VEL
LIN {X 0,Y 493.092,Z 859.31,A -85,B 0,C 180,E1 13147.061,E2 13147.061} C_VEL
LIN {X 0,Y 492.806,Z 859.31,A -85,B 0,C 180,E1 13152.429,E2 13152.429} C_VEL
LIN {X 0,Y 492.661,Z 859.31,A -85,B 0,C 180,E1 13157.911,E2 13157.911} C_VEL
LIN {X 0,Y 492.45,Z 859.31,A -85,B 0,C 180,E1 13163.575,E2 13163.575} C_VEL
LIN {X 0,Y 492.23,Z 859.31,A -85,B 0,C 180,E1 13169.502,E2 13169.502} C_VEL
LIN {X 0,Y 491.988,Z 859.31,A -85,B 0,C 180,E1 13175.808,E2 13175.808} C_VEL
LIN {X 0,Y 491.963,Z 859.31,A -85,B 0,C 180,E1 13182.334,E2 13182.334} C_VEL
LIN {X 0,Y 491.968,Z 859.31,A -85,B 0,C 180,E1 13182.982,E2 13182.982} C_VEL
LIN {X 0,Y 494.421,Z 865.035,A -85,B 0,C 180,E1 13183.387,E2 13183.387} C_VEL
LIN {X 0,Y 518.756,Z 909.863,A -85,B 0,C 180,E1 13186.742,E2 13186.742} C_VEL
LIN {X 0,Y 531.668,Z 940.895,A -85,B 0,C 180,E1 13188.642,E2 13188.642} C_VEL
LIN {X 0,Y 532.978,Z 947.702,A -85,B 0,C 180,E1 13188.966,E2 13188.966} C_VEL
LIN {X 0,Y 528.709,Z 991.609,A -85,B 0,C 180,E1 13190.407,E2 13190.407} C_VEL
LIN {X 0,Y 523.181,Z 1034.706,A -85,B 0,C 180,E1 13192.538,E2 13192.538} C_VEL
LIN {X 0,Y 516.437,Z 1076.901,A -85,B 0,C 180,E1 13195.434,E2 13195.434} C_VEL
LIN {X 0,Y 509.753,Z 1115.621,A -85,B 0,C 180,E1 13199.027,E2 13199.027} C_VEL
LIN {X 0,Y 503.682,Z 1149.459,A -85,B 0,C 180,E1 13203.175,E2 13203.175} C_VEL
LIN {X 0,Y 499.048,Z 1177.577,A -85,B 0,C 180,E1 13207.716,E2 13207.716} C_VEL
LIN {X 0,Y 496.111,Z 1198.703,A -85,B 0,C 180,E1 13212.215,E2 13212.215} C_VEL
LIN {X 0,Y 494.565,Z 1214.475,A -85,B 0,C 180,E1 13216.715,E2 13216.715} C_VEL
LIN {X 0,Y 494.083,Z 1221.444,A -85,B 0,C 180,E1 13219.392,E2 13219.392} C_VEL
LIN {X 0,Y 491.381,Z 1224.63,A -85,B 0,C 180,E1 13220.843,E2 13220.843} C_VEL
LIN {X 0,Y 485.894,Z 1228.382,A -85,B 0,C 180,E1 13223.04,E2 13223.04} C_VEL
LIN {X 0,Y 485.796,Z 1228.738,A -85,B 0,C 180,E1 13223.296,E2 13223.296} C_VEL
LIN {X 0,Y 485.73,Z 1233.205,A -85,B 0,C 180,E1 13228.212,E2 13228.212} C_VEL
LIN {X 0,Y 485.651,Z 1233.204,A -85,B 0,C 180,E1 13231.788,E2 13231.788} C_VEL
LIN {X 0,Y 485.801,Z 1229.36,A -85,B 0,C 180,E1 13236.267,E2 13236.267} C_VEL
LIN {X 0,Y 486.309,Z 1219.873,A -85,B 0,C 180,E1 13241.378,E2 13241.378} C_VEL
LIN {X 0,Y 487.646,Z 1205.337,A -85,B 0,C 180,E1 13246.24,E2 13246.24} C_VEL
LIN {X 0,Y 490.369,Z 1185.285,A -85,B 0,C 180,E1 13251.052,E2 13251.052} C_VEL
LIN {X 0,Y 494.482,Z 1159.819,A -85,B 0,C 180,E1 13255.648,E2 13255.648} C_VEL
LIN {X 0,Y 500.28,Z 1128.076,A -85,B 0,C 180,E1 13259.998,E2 13259.998} C_VEL
LIN {X 0,Y 507.117,Z 1091.181,A -85,B 0,C 180,E1 13263.828,E2 13263.828} C_VEL
LIN {X 0,Y 514.294,Z 1049.34,A -85,B 0,C 180,E1 13267.064,E2 13267.064} C_VEL
LIN {X 0,Y 520.714,Z 1005.426,A -85,B 0,C 180,E1 13269.513,E2 13269.513} C_VEL
LIN {X 0,Y 525.909,Z 958.58,A -85,B 0,C 180,E1 13271.273,E2 13271.273} C_VEL
LIN {X 0,Y 526.093,Z 945.852,A -85,B 0,C 180,E1 13271.694,E2 13271.694} C_VEL
LIN {X 0,Y 514.265,Z 915.949,A -85,B 0,C 180,E1 13273.561,E2 13273.561} C_VEL
LIN {X 0,Y 492.667,Z 875.499,A -85,B 0,C 180,E1 13276.6,E2 13276.6} C_VEL
LIN {X 0,Y 484.288,Z 860.856,A -85,B 0,C 180,E1 13277.869,E2 13277.869} C_VEL
LIN {X 0,Y 484.126,Z 859.31,A -85,B 0,C 180,E1 13278.036,E2 13278.036} C_VEL
LIN {X 0,Y 484.043,Z 859.31,A -85,B 0,C 180,E1 13284.481,E2 13284.481} C_VEL
LIN {X 0,Y 484.294,Z 859.31,A -85,B 0,C 180,E1 13289.965,E2 13289.965} C_VEL
LIN {X 0,Y 484.502,Z 859.31,A -85,B 0,C 180,E1 13296.014,E2 13296.014} C_VEL
LIN {X 0,Y 484.704,Z 859.31,A -85,B 0,C 180,E1 13301.785,E2 13301.785} C_VEL
LIN {X 0,Y 484.848,Z 859.31,A -85,B 0,C 180,E1 13307.364,E2 13307.364} C_VEL
LIN {X 0,Y 485.187,Z 859.31,A -85,B 0,C 180,E1 13312.823,E2 13312.823} C_VEL
LIN {X 0,Y 485.453,Z 859.31,A -85,B 0,C 180,E1 13318.209,E2 13318.209} C_VEL
LIN {X 0,Y 485.417,Z 859.31,A -85,B 0,C 180,E1 13323.576,E2 13323.576} C_VEL
LIN {X 0,Y 485.055,Z 859.31,A -85,B 0,C 180,E1 13328.981,E2 13328.981} C_VEL
LIN {X 0,Y 484.844,Z 859.31,A -85,B 0,C 180,E1 13334.473,E2 13334.473} C_VEL
LIN {X 0,Y 484.611,Z 859.31,A -85,B 0,C 180,E1 13340.274,E2 13340.274} C_VEL
LIN {X 0,Y 484.373,Z 859.31,A -85,B 0,C 180,E1 13345.964,E2 13345.964} C_VEL
LIN {X 0,Y 484.161,Z 859.31,A -85,B 0,C 180,E1 13352.326,E2 13352.326} C_VEL
LIN {X 0,Y 484.044,Z 859.31,A -85,B 0,C 180,E1 13358.747,E2 13358.747} C_VEL
LIN {X 0,Y 483.959,Z 859.31,A -85,B 0,C 180,E1 13363.934,E2 13363.934} C_VEL
LIN {X 0,Y 484.131,Z 859.893,A -85,B 0,C 180,E1 13368.231,E2 13368.231} C_VEL
LIN {X 0,Y 489.566,Z 870.13,A -85,B 0,C 180,E1 13369.051,E2 13369.051} C_VEL
LIN {X 0,Y 512.184,Z 909.895,A -85,B 0,C 180,E1 13372.12,E2 13372.12} C_VEL
LIN {X 0,Y 527.57,Z 941.523,A -85,B 0,C 180,E1 13374.054,E2 13374.054} C_VEL
LIN {X 0,Y 524.898,Z 984.538,A -85,B 0,C 180,E1 13374.947,E2 13374.947} C_VEL
LIN {X 0,Y 520.233,Z 1023.867,A -85,B 0,C 180,E1 13376.399,E2 13376.399} C_VEL
LIN {X 0,Y 514.25,Z 1061.102,A -85,B 0,C 180,E1 13378.481,E2 13378.481} C_VEL
LIN {X 0,Y 507.444,Z 1095.769,A -85,B 0,C 180,E1 13381.216,E2 13381.216} C_VEL
LIN {X 0,Y 500.883,Z 1125.946,A -85,B 0,C 180,E1 13384.463,E2 13384.463} C_VEL
LIN {X 0,Y 495.12,Z 1151.904,A -85,B 0,C 180,E1 13388.218,E2 13388.218} C_VEL
LIN {X 0,Y 490.626,Z 1173.436,A -85,B 0,C 180,E1 13392.442,E2 13392.442} C_VEL
LIN {X 0,Y 487.721,Z 1189.967,A -85,B 0,C 180,E1 13396.983,E2 13396.983} C_VEL
LIN {X 0,Y 486.225,Z 1201.69,A -85,B 0,C 180,E1 13401.938,E2 13401.938} C_VEL
LIN {X 0,Y 485.791,Z 1207.365,A -85,B 0,C 180,E1 13406.424,E2 13406.424} C_VEL
LIN {X 0,Y 485.702,Z 1208.734,A -85,B 0,C 180,E1 13410,E2 13410} C_VEL
LIN {X 0,Y 485.774,Z 1207.138,A -85,B 0,C 180,E1 13413.733,E2 13413.733} C_VEL
LIN {X 0,Y 486.282,Z 1201.532,A -85,B 0,C 180,E1 13418.061,E2 13418.061} C_VEL
LIN {X 0,Y 487.789,Z 1189.693,A -85,B 0,C 180,E1 13423.016,E2 13423.016} C_VEL
LIN {X 0,Y 490.645,Z 1173.021,A -85,B 0,C 180,E1 13427.566,E2 13427.566} C_VEL
LIN {X 0,Y 495.536,Z 1150.016,A -85,B 0,C 180,E1 13431.999,E2 13431.999} C_VEL
LIN {X 0,Y 501.414,Z 1123.472,A -85,B 0,C 180,E1 13435.749,E2 13435.749} C_VEL
LIN {X 0,Y 508.337,Z 1091.263,A -85,B 0,C 180,E1 13439.095,E2 13439.095} C_VEL
LIN {X 0,Y 514.892,Z 1056.941,A -85,B 0,C 180,E1 13441.697,E2 13441.697} C_VEL
LIN {X 0,Y 520.791,Z 1018.879,A -85,B 0,C 180,E1 13443.733,E2 13443.733} C_VEL
LIN {X 0,Y 525.269,Z 979.067,A -85,B 0,C 180,E1 13445.111,E2 13445.111} C_VEL
LIN {X 0,Y 526.966,Z 940.182,A -85,B 0,C 180,E1 13445.92,E2 13445.92} C_VEL
LIN {X 0,Y 504.663,Z 895.933,A -85,B 0,C 180,E1 13448.761,E2 13448.761} C_VEL
LIN {X 0,Y 484.168,Z 860.423,A -85,B 0,C 180,E1 13451.643,E2 13451.643} C_VEL
LIN {X 0,Y 484.067,Z 859.31,A -85,B 0,C 180,E1 13451.81,E2 13451.81} C_VEL
LIN {X 0,Y 483.983,Z 859.31,A -85,B 0,C 180,E1 13458.713,E2 13458.713} C_VEL
LIN {X 0,Y 484.111,Z 859.31,A -85,B 0,C 180,E1 13464.471,E2 13464.471} C_VEL
LIN {X 0,Y 484.269,Z 859.31,A -85,B 0,C 180,E1 13469.969,E2 13469.969} C_VEL
LIN {X 0,Y 484.44,Z 859.31,A -85,B 0,C 180,E1 13476.016,E2 13476.016} C_VEL
LIN {X 0,Y 484.513,Z 859.31,A -85,B 0,C 180,E1 13481.783,E2 13481.783} C_VEL
LIN {X 0,Y 484.821,Z 859.31,A -85,B 0,C 180,E1 13487.368,E2 13487.368} C_VEL
LIN {X 0,Y 485.231,Z 859.31,A -85,B 0,C 180,E1 13492.829,E2 13492.829} C_VEL
LIN {X 0,Y 485.457,Z 859.31,A -85,B 0,C 180,E1 13498.214,E2 13498.214} C_VEL
LIN {X 0,Y 485.423,Z 859.31,A -85,B 0,C 180,E1 13503.581,E2 13503.581} C_VEL
LIN {X 0,Y 485.043,Z 859.31,A -85,B 0,C 180,E1 13508.987,E2 13508.987} C_VEL
LIN {X 0,Y 484.846,Z 859.31,A -85,B 0,C 180,E1 13514.478,E2 13514.478} C_VEL
LIN {X 0,Y 484.643,Z 859.31,A -85,B 0,C 180,E1 13520.283,E2 13520.283} C_VEL
LIN {X 0,Y 484.399,Z 859.31,A -85,B 0,C 180,E1 13525.968,E2 13525.968} C_VEL
LIN {X 0,Y 484.172,Z 859.31,A -85,B 0,C 180,E1 13532.327,E2 13532.327} C_VEL
LIN {X 0,Y 484.039,Z 859.31,A -85,B 0,C 180,E1 13538.754,E2 13538.754} C_VEL
LIN {X 0,Y 484.048,Z 859.31,A -85,B 0,C 180,E1 13542.075,E2 13542.075} C_VEL
LIN {X 0,Y 486.533,Z 865.054,A -85,B 0,C 180,E1 13542.501,E2 13542.501} C_VEL
LIN {X 0,Y 511.37,Z 910.073,A -85,B 0,C 180,E1 13546.047,E2 13546.047} C_VEL
LIN {X 0,Y 525.07,Z 942.494,A -85,B 0,C 180,E1 13548.118,E2 13548.118} C_VEL
LIN {X 0,Y 526.51,Z 950.389,A -85,B 0,C 180,E1 13548.507,E2 13548.507} C_VEL
LIN {X 0,Y 522.201,Z 992.794,A -85,B 0,C 180,E1 13549.937,E2 13549.937} C_VEL
LIN {X 0,Y 516.501,Z 1035.515,A -85,B 0,C 180,E1 13552.081,E2 13552.081} C_VEL
LIN {X 0,Y 509.44,Z 1078.015,A -85,B 0,C 180,E1 13555.048,E2 13555.048} C_VEL
LIN {X 0,Y 502.54,Z 1116.216,A -85,B 0,C 180,E1 13558.658,E2 13558.658} C_VEL
LIN {X 0,Y 496.068,Z 1150.688,A -85,B 0,C 180,E1 13562.975,E2 13562.975} C_VEL
LIN {X 0,Y 491.198,Z 1179.164,A -85,B 0,C 180,E1 13567.708,E2 13567.708} C_VEL
LIN {X 0,Y 487.997,Z 1202.051,A -85,B 0,C 180,E1 13572.843,E2 13572.843} C_VEL
LIN {X 0,Y 486.401,Z 1218.303,A -85,B 0,C 180,E1 13578.015,E2 13578.015} C_VEL
LIN {X 0,Y 485.819,Z 1228.081,A -85,B 0,C 180,E1 13582.833,E2 13582.833} C_VEL
LIN {X 0,Y 485.796,Z 1228.738,A -85,B 0,C 180,E1 13583.296,E2 13583.296} C_VEL
LIN {X 0,Y 483.204,Z 1230.623,A -85,B 0,C 180,E1 13584.796,E2 13584.796} C_VEL
LIN {X 0,Y 477.809,Z 1232.384,A -85,B 0,C 180,E1 13587.059,E2 13587.059} C_VEL
LIN {X 0,Y 477.728,Z 1232.511,A -85,B 0,C 180,E1 13587.322,E2 13587.322} C_VEL
LIN {X 0,Y 477.756,Z 1233.002,A -85,B 0,C 180,E1 13591.817,E2 13591.817} C_VEL
LIN {X 0,Y 477.926,Z 1229.146,A -85,B 0,C 180,E1 13596.371,E2 13596.371} C_VEL
LIN {X 0,Y 478.421,Z 1219.969,A -85,B 0,C 180,E1 13601.417,E2 13601.417} C_VEL
LIN {X 0,Y 479.856,Z 1205.069,A -85,B 0,C 180,E1 13606.511,E2 13606.511} C_VEL
LIN {X 0,Y 482.719,Z 1184.974,A -85,B 0,C 180,E1 13611.402,E2 13611.402} C_VEL
LIN {X 0,Y 487.157,Z 1159.458,A -85,B 0,C 180,E1 13616.063,E2 13616.063} C_VEL
LIN {X 0,Y 493.001,Z 1128.457,A -85,B 0,C 180,E1 13620.379,E2 13620.379} C_VEL
LIN {X 0,Y 500.315,Z 1090.779,A -85,B 0,C 180,E1 13624.339,E2 13624.339} C_VEL
LIN {X 0,Y 507.71,Z 1049.369,A -85,B 0,C 180,E1 13627.569,E2 13627.569} C_VEL
LIN {X 0,Y 514.391,Z 1004.958,A -85,B 0,C 180,E1 13630.064,E2 13630.064} C_VEL
LIN {X 0,Y 519.709,Z 958.397,A -85,B 0,C 180,E1 13631.82,E2 13631.82} C_VEL
LIN {X 0,Y 519.79,Z 948.306,A -85,B 0,C 180,E1 13632.166,E2 13632.166} C_VEL
LIN {X 0,Y 507.607,Z 917.628,A -85,B 0,C 180,E1 13634.166,E2 13634.166} C_VEL
LIN {X 0,Y 485.415,Z 876.258,A -85,B 0,C 180,E1 13637.401,E2 13637.401} C_VEL
LIN {X 0,Y 476.299,Z 860.814,A -85,B 0,C 180,E1 13638.83,E2 13638.83} C_VEL
LIN {X 0,Y 476.168,Z 859.31,A -85,B 0,C 180,E1 13638.986,E2 13638.986} C_VEL
LIN {X 0,Y 476.178,Z 859.31,A -85,B 0,C 180,E1 13645.829,E2 13645.829} C_VEL
LIN {X 0,Y 476.415,Z 859.31,A -85,B 0,C 180,E1 13651.51,E2 13651.51} C_VEL
LIN {X 0,Y 476.645,Z 859.31,A -85,B 0,C 180,E1 13657.578,E2 13657.578} C_VEL
LIN {X 0,Y 476.825,Z 859.31,A -85,B 0,C 180,E1 13663.383,E2 13663.383} C_VEL
LIN {X 0,Y 477.067,Z 859.31,A -85,B 0,C 180,E1 13669.944,E2 13669.944} C_VEL
LIN {X 0,Y 477.528,Z 859.31,A -85,B 0,C 180,E1 13676.36,E2 13676.36} C_VEL
LIN {X 0,Y 477.644,Z 859.31,A -85,B 0,C 180,E1 13681.815,E2 13681.815} C_VEL
LIN {X 0,Y 477.252,Z 859.31,A -85,B 0,C 180,E1 13687.292,E2 13687.292} C_VEL
LIN {X 0,Y 476.983,Z 859.31,A -85,B 0,C 180,E1 13692.843,E2 13692.843} C_VEL
LIN {X 0,Y 476.754,Z 859.31,A -85,B 0,C 180,E1 13698.524,E2 13698.524} C_VEL
LIN {X 0,Y 476.505,Z 859.31,A -85,B 0,C 180,E1 13704.409,E2 13704.409} C_VEL
LIN {X 0,Y 476.259,Z 859.31,A -85,B 0,C 180,E1 13710.791,E2 13710.791} C_VEL
LIN {X 0,Y 476.09,Z 859.31,A -85,B 0,C 180,E1 13717.279,E2 13717.279} C_VEL
LIN {X 0,Y 476.001,Z 859.31,A -85,B 0,C 180,E1 13722.931,E2 13722.931} C_VEL
LIN {X 0,Y 476.199,Z 859.31,A -85,B 0,C 180,E1 13727.241,E2 13727.241} C_VEL
LIN {X 0,Y 478.709,Z 865.083,A -85,B 0,C 180,E1 13727.679,E2 13727.679} C_VEL
LIN {X 0,Y 503.271,Z 907.397,A -85,B 0,C 180,E1 13731.187,E2 13731.187} C_VEL
LIN {X 0,Y 521.382,Z 944.959,A -85,B 0,C 180,E1 13733.565,E2 13733.565} C_VEL
